KUKA KRL program: MyProgram_225().src

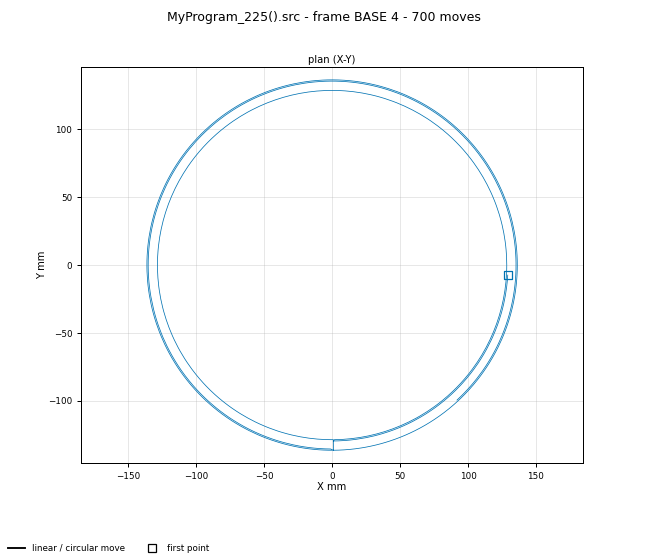
[picture p0: tool path of MyProgram_225().src in frame BASE 4, 700 of 700 moves have a stored position in this frame; points joined in program order, loops and branches not executed]
&ACCESS RVP
&REL 1
&PARAM TEMPLATE = C:\KRC\Roboter\Template\vorgabe
&PARAM EDITMASK = *
DEF MyProgram_225()
; ---- Setting reference (Base) ----
$BASE = BASE_DATA[4]

; --------------------------
; ---- Setting tool (TCP) ----
$TOOL = TOOL_DATA[3]
; --------------------------

$VEL.CP = VEL_APROX_PRINT
Startdeposition()
$VEL.CP = VEL_PRINT
LIN {X 129.2474,Y -7.3831,Z 155,A -4.9657,B 16.1496,C -0.2216,E1 16.3104,E2 814.1101} C_DIS
LIN {X 128.9531,Y -11.421,Z 155,A -6.9054,B 16.1497,C -0.211,E1 16.3099,E2 816.0693} C_DIS
LIN {X 128.4281,Y -16.2953,Z 155,A -8.4504,B 16.1495,C -0.2265,E1 16.3095,E2 817.5445} C_DIS
LIN {X 127.4709,Y -22.5885,Z 155,A -10.9683,B 16.1495,C -0.2286,E1 16.3084,E2 820.031} C_DIS
LIN {X 127.0051,Y -25.0853,Z 155,A -12.6562,B 16.1498,C -0.2051,E1 16.3075,E2 821.7867} C_DIS
LIN {X 126.3261,Y -28.3023,Z 155,A -13.8755,B 16.1498,C -0.2091,E1 16.3067,E2 822.9803} C_DIS
LIN {X 125.3243,Y -32.4531,Z 155,A -15.5909,B 16.1498,C -0.2097,E1 16.3056,E2 824.678} C_DIS
LIN {X 124.4903,Y -35.5191,Z 155,A -17.2829,B 16.1499,C -0.1954,E1 16.3043,E2 826.4054} C_DIS
LIN {X 122.9714,Y -40.4627,Z 155,A -19.3134,B 16.1499,C -0.1978,E1 16.3026,E2 828.4087} C_DIS
LIN {X 121.7271,Y -44.0625,Z 155,A -21.5995,B 16.1502,C -0.1717,E1 16.3004,E2 830.7672} C_DIS
LIN {X 119.9725,Y -48.6377,Z 155,A -23.157,B 16.15,C -0.187,E1 16.2988,E2 832.2564} C_DIS
LIN {X 118.5111,Y -52.1027,Z 155,A -24.7542,B 16.15,C -0.1846,E1 16.2971,E2 833.8481} C_DIS
LIN {X 117.1159,Y -55.1662,Z 155,A -26.2187,B 16.15,C -0.1813,E1 16.2954,E2 835.3116} C_DIS
LIN {X 114.7718,Y -59.8872,Z 155,A -28.3572,B 16.15,C -0.1817,E1 16.2927,E2 837.4305} C_DIS
LIN {X 113.6651,Y -61.9653,Z 155,A -29.6574,B 16.1502,C -0.1696,E1 16.2909,E2 838.7625} C_DIS
LIN {X 111.4503,Y -65.8666,Z 155,A -31.6784,B 16.1502,C -0.163,E1 16.2881,E2 840.7904} C_DIS
LIN {X 109.1625,Y -69.5921,Z 155,A -33.4546,B 16.1502,C -0.1634,E1 16.2855,E2 842.5506} C_DIS
LIN {X 107.339,Y -72.3729,Z 155,A -35.0483,B 16.1503,C -0.1553,E1 16.283,E2 844.1606} C_DIS
LIN {X 104.186,Y -76.8426,Z 155,A -37.4354,B 16.1503,C -0.1503,E1 16.2791,E2 846.547} C_DIS
LIN {X 101.853,Y -79.9088,Z 155,A -39.1319,B 16.1504,C -0.1463,E1 16.2762,E2 848.2447} C_DIS
LIN {X 99.343,Y -83.0089,Z 155,A -40.9388,B 16.1504,C -0.1406,E1 16.273,E2 850.0588} C_DIS
LIN {X 96.0502,Y -86.7978,Z 155,A -42.9236,B 16.1504,C -0.1435,E1 16.2694,E2 852.0187} C_DIS
LIN {X 93.7861,Y -89.2396,Z 155,A -44.5289,B 16.1505,C -0.1355,E1 16.2663,E2 853.6413} C_DIS
LIN {X 90.8438,Y -92.233,Z 155,A -46.4781,B 16.1505,C -0.1281,E1 16.2624,E2 855.6036} C_DIS
LIN {X 87.5864,Y -95.3314,Z 155,A -48.1246,B 16.1505,C -0.1357,E1 16.2591,E2 857.2121} C_DIS
LIN {X 85.2485,Y -97.4277,Z 155,A -49.6523,B 16.1505,C -0.1279,E1 16.2559,E2 858.7578} C_DIS
LIN {X 82.2321,Y -99.9874,Z 155,A -51.4278,B 16.1505,C -0.1234,E1 16.2521,E2 860.5383} C_DIS
LIN {X 78.358,Y -103.0515,Z 155,A -53.5577,B 16.1506,C -0.121,E1 16.2474,E2 862.6642} C_DIS
LIN {X 75.3005,Y -105.3056,Z 155,A -55.2753,B 16.1506,C -0.1165,E1 16.2435,E2 864.388} C_DIS
LIN {X 71.8133,Y -107.714,Z 155,A -57.181,B 16.1506,C -0.112,E1 16.2391,E2 866.2994} C_DIS
LIN {X 68.6345,Y -109.7672,Z 155,A -58.8635,B 16.1507,C -0.1088,E1 16.2351,E2 867.9846} C_DIS
LIN {X 64.898,Y -112.0165,Z 155,A -60.7724,B 16.1507,C -0.1063,E1 16.2305,E2 869.8931} C_DIS
LIN {X 59.3003,Y -115.0774,Z 155,A -63.965,B 16.1508,C -0.0893,E1 16.2226,E2 873.1319} C_DIS
LIN {X 55.719,Y -116.8518,Z 155,A -65.2781,B 16.1508,C -0.1022,E1 16.2194,E2 874.3933} C_DIS
LIN {X 52.249,Y -118.4459,Z 155,A -67.4256,B 16.1508,C -0.0844,E1 16.2138,E2 876.596} C_DIS
LIN {X 48.4916,Y -120.0314,Z 155,A -68.8253,B 16.1508,C -0.0957,E1 16.2103,E2 877.9501} C_DIS
LIN {X 45.0598,Y -121.3619,Z 155,A -70.3403,B 16.1508,C -0.0975,E1 16.2063,E2 879.4531} C_DIS
LIN {X 41.6197,Y -122.5861,Z 155,A -72.6412,B 16.1508,C -0.0727,E1 16.2001,E2 881.8356} C_DIS
LIN {X 36.809,Y -124.114,Z 155,A -74.0346,B 16.1508,C -0.0985,E1 16.1966,E2 883.1326} C_DIS
LIN {X 33.8596,Y -124.9512,Z 155,A -75.564,B 16.1508,C -0.0914,E1 16.1924,E2 884.6834} C_DIS
LIN {X 30.5927,Y -125.7901,Z 155,A -77.8519,B 16.1509,C -0.0637,E1 16.186,E2 887.0651} C_DIS
LIN {X 24.8487,Y -127.0506,Z 155,A -79.6789,B 16.1509,C -0.0873,E1 16.1812,E2 888.8038} C_DIS
LIN {X 17.4336,Y -128.279,Z 155,A -82.8576,B 16.1509,C -0.0901,E1 16.1725,E2 891.9675} C_DIS
LIN {X 13.1784,Y -128.786,Z 155,A -84.9822,B 16.1509,C -0.0816,E1 16.1665,E2 894.12} C_DIS
LIN {X 9.2675,Y -129.1248,Z 155,A -86.6956,B 16.1509,C -0.0817,E1 16.1617,E2 895.8316} C_DIS
LIN {X 4.804,Y -129.3679,Z 155,A -88.6412,B 16.1509,C -0.0822,E1 16.1563,E2 897.7745} C_DIS
LIN {X 0.918,Y -129.4524,Z 155,A -89.6672,B 16.1507,C -0.1046,E1 16.1537,E2 898.7195} C_DIS
Enddeposition()
LIN {X 0.918,Y -129.4524,Z 155,A -89.6672,B 16.1507,C -0.1046,E1 16.1537,E2 898.7195} C_DIS
Startdeposition()
$VEL.CP = VEL_PRINT
LIN {X 1.6778,Y -128.5115,Z 155,A -89.2328,B 16.1506,C -0.1179,E1 16.1549,E2 898.2373} C_DIS
LIN {X 4.7325,Y -128.4347,Z 155,A -87.9227,B 16.1506,C -0.1166,E1 16.1586,E2 896.9326} C_DIS
LIN {X 7.9871,Y -128.2732,Z 155,A -86.5233,B 16.1506,C -0.1153,E1 16.1625,E2 895.5387} C_DIS
LIN {X 11.132,Y -128.0389,Z 155,A -85.1192,B 16.1506,C -0.1158,E1 16.1664,E2 894.134} C_DIS
LIN {X 14.3466,Y -127.7196,Z 155,A -83.6808,B 16.1506,C -0.1165,E1 16.1704,E2 892.6949} C_DIS
LIN {X 17.4169,Y -127.3379,Z 155,A -82.2994,B 16.1506,C -0.1173,E1 16.1742,E2 891.3124} C_DIS
LIN {X 20.4129,Y -126.8922,Z 155,A -80.9516,B 16.1506,C -0.118,E1 16.1779,E2 889.964} C_DIS
LIN {X 23.6323,Y -126.331,Z 155,A -79.5141,B 16.1506,C -0.1184,E1 16.1819,E2 888.5277} C_DIS
LIN {X 26.7059,Y -125.7168,Z 155,A -78.0866,B 16.1506,C -0.1205,E1 16.1858,E2 887.0956} C_DIS
LIN {X 30.0992,Y -124.947,Z 155,A -76.4897,B 16.1506,C -0.1234,E1 16.1902,E2 885.4921} C_DIS
LIN {X 32.8535,Y -124.2515,Z 155,A -75.2461,B 16.1506,C -0.1238,E1 16.1935,E2 884.2502} C_DIS
LIN {X 35.7824,Y -123.4401,Z 155,A -73.9279,B 16.1506,C -0.1238,E1 16.197,E2 882.9352} C_DIS
LIN {X 38.7952,Y -122.5265,Z 155,A -72.5303,B 16.1506,C -0.1252,E1 16.2008,E2 881.537} C_DIS
LIN {X 42.2001,Y -121.3954,Z 155,A -71.0011,B 16.1506,C -0.1246,E1 16.2048,E2 880.0147} C_DIS
LIN {X 44.8787,Y -120.431,Z 155,A -69.6719,B 16.1505,C -0.1282,E1 16.2083,E2 878.6774} C_DIS
LIN {X 47.8161,Y -119.2953,Z 155,A -68.2677,B 16.1505,C -0.13,E1 16.212,E2 877.2717} C_DIS
LIN {X 50.745,Y -118.0792,Z 155,A -66.9012,B 16.1505,C -0.1302,E1 16.2155,E2 875.9094} C_DIS
LIN {X 53.6147,Y -116.8044,Z 155,A -65.477,B 16.1505,C -0.133,E1 16.2191,E2 874.481} C_DIS
LIN {X 56.4616,Y -115.4553,Z 155,A -64.0855,B 16.1505,C -0.1346,E1 16.2226,E2 873.0897} C_DIS
LIN {X 59.1544,Y -114.1002,Z 155,A -62.7618,B 16.1505,C -0.136,E1 16.2259,E2 871.767} C_DIS
LIN {X 61.9121,Y -112.6286,Z 155,A -61.238,B 16.1504,C -0.1427,E1 16.2297,E2 870.2265} C_DIS
LIN {X 64.7163,Y -111.041,Z 155,A -59.8975,B 16.1504,C -0.1417,E1 16.2329,E2 868.8957} C_DIS
LIN {X 67.5215,Y -109.3579,Z 155,A -58.4653,B 16.1504,C -0.1433,E1 16.2363,E2 867.4651} C_DIS
LIN {X 70.18,Y -107.6707,Z 155,A -57.0713,B 16.1504,C -0.1455,E1 16.2396,E2 866.0706} C_DIS
LIN {X 72.7088,Y -105.9792,Z 155,A -55.7279,B 16.1504,C -0.1476,E1 16.2427,E2 864.7272} C_DIS
LIN {X 75.3703,Y -104.1032,Z 155,A -54.2861,B 16.1504,C -0.15,E1 16.2459,E2 863.2849} C_DIS
LIN {X 78.4386,Y -101.812,Z 155,A -52.4335,B 16.1502,C -0.1584,E1 16.2501,E2 861.4131} C_DIS
LIN {X 81.5351,Y -99.3492,Z 155,A -50.6751,B 16.1502,C -0.1618,E1 16.2539,E2 859.6532} C_DIS
LIN {X 85.1286,Y -96.2875,Z 155,A -48.5905,B 16.1502,C -0.1656,E1 16.2583,E2 857.5684} C_DIS
LIN {X 88.6071,Y -93.0967,Z 155,A -46.5125,B 16.1502,C -0.1692,E1 16.2626,E2 855.4909} C_DIS
LIN {X 91.4722,Y -90.2838,Z 155,A -44.7234,B 16.1501,C -0.1733,E1 16.2661,E2 853.6997} C_DIS
LIN {X 94.6884,Y -86.9039,Z 155,A -42.6573,B 16.1501,C -0.1776,E1 16.27,E2 851.6326} C_DIS
LIN {X 97.8259,Y -83.3563,Z 155,A -40.5635,B 16.15,C -0.1821,E1 16.2739,E2 849.5381} C_DIS
LIN {X 100.8306,Y -79.6963,Z 155,A -38.4709,B 16.15,C -0.1866,E1 16.2775,E2 847.445} C_DIS
LIN {X 103.2224,Y -76.5725,Z 155,A -36.8644,B 16.15,C -0.1858,E1 16.2802,E2 845.8536} C_DIS
LIN {X 105.4013,Y -73.5443,Z 155,A -35.3387,B 16.15,C -0.1853,E1 16.2827,E2 844.3419} C_DIS
LIN {X 106.8625,Y -71.4043,Z 155,A -34.0899,B 16.1499,C -0.1916,E1 16.2846,E2 843.0805} C_DIS
LIN {X 108.5817,Y -68.7621,Z 155,A -32.6993,B 16.1499,C -0.1948,E1 16.2867,E2 841.6896} C_DIS
LIN {X 110.2875,Y -65.9916,Z 155,A -31.1326,B 16.1498,C -0.2028,E1 16.289,E2 840.1073} C_DIS
LIN {X 111.8819,Y -63.2511,Z 155,A -29.8604,B 16.1498,C -0.2016,E1 16.2908,E2 838.8498} C_DIS
LIN {X 113.3987,Y -60.4901,Z 155,A -28.4494,B 16.1498,C -0.2057,E1 16.2926,E2 837.4361} C_DIS
LIN {X 114.8075,Y -57.769,Z 155,A -27.1034,B 16.1497,C -0.2088,E1 16.2943,E2 836.0906} C_DIS
LIN {X 116.1854,Y -54.9443,Z 155,A -25.6971,B 16.1497,C -0.2129,E1 16.296,E2 834.6817} C_DIS
LIN {X 117.4948,Y -52.0848,Z 155,A -24.329,B 16.1496,C -0.2157,E1 16.2976,E2 833.3156} C_DIS
LIN {X 118.734,Y -49.194,Z 155,A -22.9407,B 16.1496,C -0.2192,E1 16.2991,E2 831.927} C_DIS
LIN {X 119.9017,Y -46.2748,Z 155,A -21.5531,B 16.1495,C -0.2228,E1 16.3005,E2 830.5392} C_DIS
LIN {X 121.0454,Y -43.1959,Z 155,A -20.102,B 16.1495,C -0.2266,E1 16.3019,E2 829.0876} C_DIS
LIN {X 122.0688,Y -40.2129,Z 155,A -18.7106,B 16.1494,C -0.2302,E1 16.3031,E2 827.696} C_DIS
LIN {X 123.0231,Y -37.1916,Z 155,A -17.3224,B 16.1494,C -0.2335,E1 16.3043,E2 826.3087} C_DIS
LIN {X 123.8678,Y -34.2723,Z 155,A -15.9674,B 16.1493,C -0.2375,E1 16.3053,E2 824.9518} C_DIS
LIN {X 124.6966,Y -31.1243,Z 155,A -14.5432,B 16.1493,C -0.2409,E1 16.3063,E2 823.5288} C_DIS
LIN {X 125.398,Y -28.1654,Z 155,A -13.1855,B 16.1492,C -0.245,E1 16.3072,E2 822.169} C_DIS
LIN {X 126.0535,Y -25.0714,Z 155,A -11.7956,B 16.1492,C -0.2485,E1 16.3079,E2 820.7795} C_DIS
LIN {X 126.6293,Y -21.9819,Z 155,A -10.4121,B 16.1491,C -0.2521,E1 16.3086,E2 819.3962} C_DIS
LIN {X 127.1333,Y -18.8507,Z 155,A -8.9602,B 16.149,C -0.2578,E1 16.3092,E2 817.9379} C_DIS
LIN {X 127.5546,Y -15.7436,Z 155,A -7.5816,B 16.149,C -0.2613,E1 16.3097,E2 816.5597} C_DIS
LIN {X 127.9003,Y -12.6262,Z 155,A -6.2052,B 16.1489,C -0.2648,E1 16.3101,E2 815.184} C_DIS
LIN {X 128.1695,Y -9.507,Z 155,A -4.852,B 16.1489,C -0.2676,E1 16.3104,E2 813.8339} C_DIS
LIN {X 128.3721,Y -6.2015,Z 155,A -3.3818,B 16.1488,C -0.2718,E1 16.3107,E2 812.3625} C_DIS
LIN {X 128.4838,Y -3.1456,Z 155,A -2.0505,B 16.1488,C -0.2748,E1 16.3107,E2 811.0332} C_DIS
LIN {X 128.5245,Y 0.0068,Z 155,A -0.4873,B 16.1486,C -0.2847,E1 16.3107,E2 809.4497} C_DIS
LIN {X 128.4806,Y 3.2619,Z 155,A 0.7946,B 16.1486,C -0.2831,E1 16.3107,E2 808.1858} C_DIS
LIN {X 128.3589,Y 6.4648,Z 155,A 2.2721,B 16.1485,C -0.2892,E1 16.3105,E2 806.7007} C_DIS
LIN {X 128.0428,Y 11.0858,Z 155,A 4.2244,B 16.1485,C -0.2914,E1 16.3101,E2 804.7591} C_DIS
LIN {X 127.7458,Y 14.1038,Z 155,A 5.7395,B 16.1483,C -0.3013,E1 16.3097,E2 803.2231} C_DIS
LIN {X 127.3364,Y 17.4282,Z 155,A 7.0732,B 16.1483,C -0.3001,E1 16.3092,E2 801.9065} C_DIS
LIN {X 126.8629,Y 20.5886,Z 155,A 8.5421,B 16.1482,C -0.3059,E1 16.3085,E2 800.4307} C_DIS
LIN {X 126.3334,Y 23.6197,Z 155,A 9.8059,B 16.1482,C -0.3062,E1 16.3079,E2 799.1778} C_DIS
LIN {X 125.7187,Y 26.6971,Z 155,A 11.225,B 16.1481,C -0.311,E1 16.3071,E2 797.7547} C_DIS
LIN {X 125.0528,Y 29.6603,Z 155,A 12.6772,B 16.1479,C -0.3185,E1 16.3062,E2 796.2895} C_DIS
LIN {X 124.0111,Y 33.7549,Z 155,A 14.5681,B 16.1479,C -0.3242,E1 16.3048,E2 794.3957} C_DIS
LIN {X 122.9892,Y 37.3025,Z 155,A 16.0644,B 16.1479,C -0.3237,E1 16.3037,E2 792.915} C_DIS
LIN {X 122.0342,Y 40.3168,Z 155,A 17.4933,B 16.1477,C -0.3284,E1 16.3024,E2 791.4823} C_DIS
LIN {X 120.9718,Y 43.3998,Z 155,A 18.8986,B 16.1477,C -0.3308,E1 16.3011,E2 790.0811} C_DIS
LIN {X 119.8705,Y 46.3552,Z 155,A 20.2903,B 16.1477,C -0.3342,E1 16.2997,E2 788.6896} C_DIS
LIN {X 118.397,Y 50.001,Z 155,A 22.1728,B 16.1474,C -0.3436,E1 16.2977,E2 786.7902} C_DIS
LIN {X 116.81,Y 53.6026,Z 155,A 23.7609,B 16.1474,C -0.3425,E1 16.2959,E2 785.2198} C_DIS
LIN {X 115.4748,Y 56.4221,Z 155,A 25.2247,B 16.1474,C -0.3488,E1 16.2941,E2 783.7462} C_DIS
LIN {X 114.0834,Y 59.1864,Z 155,A 26.4948,B 16.1474,C -0.3486,E1 16.2925,E2 782.4876} C_DIS
LIN {X 112.594,Y 61.9747,Z 155,A 27.9079,B 16.1473,C -0.3525,E1 16.2906,E2 781.0728} C_DIS
LIN {X 111.041,Y 64.7163,Z 155,A 29.3254,B 16.1472,C -0.3565,E1 16.2887,E2 779.6526} C_DIS
LIN {X 109.0767,Y 67.9739,Z 155,A 30.8966,B 16.1472,C -0.3565,E1 16.2864,E2 778.0945} C_DIS
LIN {X 107.6796,Y 70.1663,Z 155,A 32.139,B 16.147,C -0.3623,E1 16.2845,E2 776.8415} C_DIS
LIN {X 106.0025,Y 72.6749,Z 155,A 33.4662,B 16.147,C -0.3649,E1 16.2824,E2 775.5152} C_DIS
LIN {X 104.1598,Y 75.2922,Z 155,A 35.0142,B 16.1468,C -0.3726,E1 16.2799,E2 773.9521} C_DIS
LIN {X 101.8049,Y 78.4478,Z 155,A 36.7885,B 16.1468,C -0.3773,E1 16.2769,E2 772.1743} C_DIS
LIN {X 99.345,Y 81.5402,Z 155,A 38.5399,B 16.1466,C -0.381,E1 16.2738,E2 770.4229} C_DIS
LIN {X 96.7667,Y 84.5835,Z 155,A 40.291,B 16.1466,C -0.384,E1 16.2706,E2 768.6738} C_DIS
LIN {X 94.1318,Y 87.5065,Z 155,A 42.0259,B 16.1465,C -0.3872,E1 16.2673,E2 766.94} C_DIS
LIN {X 90.9193,Y 90.8404,Z 155,A 43.9575,B 16.1465,C -0.3869,E1 16.2636,E2 765.0225} C_DIS
LIN {X 88.0408,Y 93.6324,Z 155,A 45.8629,B 16.1463,C -0.3946,E1 16.2597,E2 763.1025} C_DIS
LIN {X 85.1331,Y 96.2835,Z 155,A 47.6115,B 16.1463,C -0.3978,E1 16.2561,E2 761.3538} C_DIS
LIN {X 81.5387,Y 99.3462,Z 155,A 49.7011,B 16.1461,C -0.4012,E1 16.2516,E2 759.265} C_DIS
LIN {X 77.8639,Y 102.2519,Z 155,A 51.7741,B 16.1461,C -0.4043,E1 16.247,E2 757.193} C_DIS
LIN {X 75.2011,Y 104.2259,Z 155,A 53.1006,B 16.1461,C -0.4017,E1 16.2441,E2 755.8833} C_DIS
LIN {X 72.7118,Y 105.9772,Z 155,A 54.4455,B 16.1461,C -0.4036,E1 16.241,E2 754.5394} C_DIS
LIN {X 70.092,Y 107.7279,Z 155,A 55.8445,B 16.1461,C -0.4056,E1 16.2377,E2 753.1406} C_DIS
LIN {X 67.1684,Y 109.5745,Z 155,A 57.3256,B 16.1461,C -0.4059,E1 16.2342,E2 751.666} C_DIS
LIN {X 64.6725,Y 111.0664,Z 155,A 58.6546,B 16.146,C -0.4089,E1 16.231,E2 750.3329} C_DIS
LIN {X 61.9909,Y 112.585,Z 155,A 60.0556,B 16.1459,C -0.4117,E1 16.2276,E2 748.9285} C_DIS
LIN {X 59.1897,Y 114.0817,Z 155,A 61.4531,B 16.1459,C -0.4129,E1 16.2241,E2 747.5329} C_DIS
LIN {X 56.3717,Y 115.4997,Z 155,A 62.8516,B 16.1459,C -0.4144,E1 16.2206,E2 746.1351} C_DIS
LIN {X 53.4283,Y 116.8906,Z 155,A 64.4625,B 16.1456,C -0.4215,E1 16.2165,E2 744.5056} C_DIS
LIN {X 50.3552,Y 118.2477,Z 155,A 65.7823,B 16.1457,C -0.4172,E1 16.2132,E2 743.2063} C_DIS
LIN {X 47.7503,Y 119.3218,Z 155,A 67.0354,B 16.1457,C -0.4184,E1 16.2099,E2 741.9534} C_DIS
LIN {X 44.849,Y 120.4422,Z 155,A 68.4256,B 16.1457,C -0.4199,E1 16.2063,E2 740.5628} C_DIS
LIN {X 41.711,Y 121.565,Z 155,A 69.9001,B 16.1457,C -0.4208,E1 16.2024,E2 739.0897} C_DIS
LIN {X 38.7098,Y 122.5538,Z 155,A 71.3037,B 16.1457,C -0.4218,E1 16.1987,E2 737.6867} C_DIS
LIN {X 35.5655,Y 123.5035,Z 155,A 72.7486,B 16.1457,C -0.4223,E1 16.1948,E2 736.2442} C_DIS
LIN {X 32.2348,Y 124.4148,Z 155,A 74.4562,B 16.1455,C -0.4289,E1 16.1902,E2 734.5175} C_DIS
LIN {X 28.1665,Y 125.3977,Z 155,A 76.1659,B 16.1455,C -0.4249,E1 16.1856,E2 732.826} C_DIS
LIN {X 25.0874,Y 126.0502,Z 155,A 77.5622,B 16.1455,C -0.4253,E1 16.1818,E2 731.4308} C_DIS
LIN {X 21.9616,Y 126.633,Z 155,A 78.9684,B 16.1455,C -0.4256,E1 16.1779,E2 730.0263} C_DIS
LIN {X 18.8606,Y 127.1318,Z 155,A 80.4238,B 16.1455,C -0.4279,E1 16.1739,E2 728.5649} C_DIS
LIN {X 15.7531,Y 127.5535,Z 155,A 81.8154,B 16.1455,C -0.4281,E1 16.17,E2 727.1745} C_DIS
LIN {X 12.6343,Y 127.8995,Z 155,A 83.2064,B 16.1455,C -0.4281,E1 16.1662,E2 725.7848} C_DIS
LIN {X 9.5076,Y 128.1695,Z 155,A 84.6793,B 16.1455,C -0.4307,E1 16.162,E2 724.304} C_DIS
LIN {X 4.7612,Y 128.4336,Z 155,A 86.6769,B 16.1455,C -0.4268,E1 16.1565,E2 722.3212} C_DIS
LIN {X 1.5922,Y 128.5129,Z 155,A 88.0233,B 16.1455,C -0.4246,E1 16.1528,E2 720.9832} C_DIS
LIN {X -1.6807,Y 128.5115,Z 155,A 89.5801,B 16.1455,C -0.4276,E1 16.1484,E2 719.4159} C_DIS
LIN {X -4.7248,Y 128.435,Z 155,A 91.0568,B 16.1454,C -0.4311,E1 16.1442,E2 717.9262} C_DIS
LIN {X -8.3936,Y 128.2481,Z 155,A 92.51,B 16.1456,C -0.4248,E1 16.1402,E2 716.495} C_DIS
LIN {X -11.1743,Y 128.0353,Z 155,A 93.7856,B 16.1456,C -0.4254,E1 16.1367,E2 715.2165} C_DIS
LIN {X -14.2979,Y 127.7249,Z 155,A 95.1896,B 16.1456,C -0.4249,E1 16.1328,E2 713.8128} C_DIS
LIN {X -17.4144,Y 127.3382,Z 155,A 96.7612,B 16.1454,C -0.4296,E1 16.1284,E2 712.2225} C_DIS
LIN {X -20.5195,Y 126.8744,Z 155,A 98.0601,B 16.1455,C -0.4256,E1 16.1248,E2 710.9361} C_DIS
LIN {X -23.6138,Y 126.3345,Z 155,A 99.3856,B 16.1456,C -0.4224,E1 16.1212,E2 709.62} C_DIS
LIN {X -26.7229,Y 125.7131,Z 155,A 100.8372,B 16.1456,C -0.4226,E1 16.1172,E2 708.1651} C_DIS
LIN {X -29.6889,Y 125.0459,Z 155,A 102.2295,B 16.1456,C -0.4226,E1 16.1134,E2 706.7697} C_DIS
LIN {X -32.86,Y 124.2498,Z 155,A 103.6553,B 16.1456,C -0.4204,E1 16.1096,E2 705.3486} C_DIS
LIN {X -35.7921,Y 123.4372,Z 155,A 105.0154,B 16.1456,C -0.4192,E1 16.1059,E2 703.9891} C_DIS
LIN {X -38.806,Y 122.523,Z 155,A 106.4232,B 16.1457,C -0.418,E1 16.1022,E2 702.5821} C_DIS
LIN {X -41.7983,Y 121.5348,Z 155,A 107.8642,B 16.1457,C -0.4176,E1 16.0984,E2 701.1382} C_DIS
LIN {X -44.8793,Y 120.4308,Z 155,A 109.2974,B 16.1458,C -0.4151,E1 16.0946,E2 699.7092} C_DIS
LIN {X -47.8351,Y 119.2876,Z 155,A 110.714,B 16.1458,C -0.4135,E1 16.0909,E2 698.2935} C_DIS
LIN {X -50.7426,Y 118.0802,Z 155,A 112.09,B 16.1459,C -0.4109,E1 16.0874,E2 696.922} C_DIS
LIN {X -53.6201,Y 116.8019,Z 155,A 113.6569,B 16.1459,C -0.4139,E1 16.0834,E2 695.3378} C_DIS
LIN {X -56.4654,Y 115.4535,Z 155,A 114.9395,B 16.1459,C -0.4083,E1 16.0802,E2 694.0705} C_DIS
LIN {X -59.1815,Y 114.086,Z 155,A 116.283,B 16.146,C -0.4059,E1 16.0769,E2 692.7297} C_DIS
LIN {X -61.9561,Y 112.6043,Z 155,A 117.7111,B 16.146,C -0.4045,E1 16.0734,E2 691.3001} C_DIS
LIN {X -65.2941,Y 110.7019,Z 155,A 119.334,B 16.1462,C -0.399,E1 16.0695,E2 689.6892} C_DIS
LIN {X -67.5233,Y 109.3567,Z 155,A 120.6102,B 16.1462,C -0.4005,E1 16.0664,E2 688.4012} C_DIS
LIN {X -70.1807,Y 107.6703,Z 155,A 122.0204,B 16.1462,C -0.3983,E1 16.0631,E2 686.9917} C_DIS
LIN {X -72.7105,Y 105.9781,Z 155,A 123.3807,B 16.1462,C -0.396,E1 16.0599,E2 685.6326} C_DIS
LIN {X -75.3746,Y 104.1001,Z 155,A 124.8414,B 16.1463,C -0.3935,E1 16.0566,E2 684.1726} C_DIS
LIN {X -78.4549,Y 101.7994,Z 155,A 126.7263,B 16.1463,C -0.3953,E1 16.0524,E2 682.2702} C_DIS
LIN {X -82.1023,Y 98.8807,Z 155,A 128.6844,B 16.1465,C -0.3874,E1 16.0482,E2 680.3288} C_DIS
LIN {X -85.1338,Y 96.2829,Z 155,A 130.6129,B 16.1465,C -0.3882,E1 16.0441,E2 678.3855} C_DIS
LIN {X -88.616,Y 93.0883,Z 155,A 132.7189,B 16.1465,C -0.3836,E1 16.0398,E2 676.2821} C_DIS
LIN {X -91.4742,Y 90.2818,Z 155,A 134.533,B 16.1466,C -0.3804,E1 16.0362,E2 674.4671} C_DIS
LIN {X -94.6944,Y 86.8973,Z 155,A 136.6338,B 16.1467,C -0.3762,E1 16.0322,E2 672.3668} C_DIS
LIN {X -97.8335,Y 83.3474,Z 155,A 138.7579,B 16.1468,C -0.3715,E1 16.0283,E2 670.2442} C_DIS
LIN {X -100.8339,Y 79.6922,Z 155,A 140.8828,B 16.1469,C -0.3669,E1 16.0246,E2 668.1201} C_DIS
LIN {X -103.6736,Y 75.9603,Z 155,A 142.9652,B 16.1471,C -0.3614,E1 16.0211,E2 666.0414} C_DIS
LIN {X -105.981,Y 72.7062,Z 155,A 144.6287,B 16.1472,C -0.3535,E1 16.0185,E2 664.3933} C_DIS
LIN {X -107.7317,Y 70.0861,Z 155,A 146.0428,B 16.1472,C -0.3501,E1 16.0163,E2 662.98} C_DIS
LIN {X -109.4371,Y 67.3924,Z 155,A 147.5003,B 16.1474,C -0.3474,E1 16.0142,E2 661.5204} C_DIS
LIN {X -111.0995,Y 64.6152,Z 155,A 148.9274,B 16.1474,C -0.3431,E1 16.0122,E2 660.097} C_DIS
LIN {X -112.6399,Y 61.8916,Z 155,A 150.3436,B 16.1475,C -0.3399,E1 16.0102,E2 658.6802} C_DIS
LIN {X -114.0659,Y 59.2198,Z 155,A 151.7105,B 16.1475,C -0.3367,E1 16.0085,E2 657.3133} C_DIS
LIN {X -115.472,Y 56.4279,Z 155,A 153.1143,B 16.1476,C -0.3332,E1 16.0067,E2 655.9101} C_DIS
LIN {X -116.9071,Y 53.3926,Z 155,A 154.6176,B 16.1477,C -0.3292,E1 16.005,E2 654.4082} C_DIS
LIN {X -118.1251,Y 50.6389,Z 155,A 155.978,B 16.1477,C -0.3259,E1 16.0034,E2 653.0476} C_DIS
LIN {X -119.3315,Y 47.7262,Z 155,A 157.3951,B 16.1479,C -0.3222,E1 16.002,E2 651.631} C_DIS
LIN {X -120.4648,Y 44.7886,Z 155,A 158.9725,B 16.1479,C -0.3232,E1 16.0004,E2 650.0357} C_DIS
LIN {X -121.571,Y 41.6936,Z 155,A 160.2898,B 16.148,C -0.3146,E1 15.9992,E2 648.7374} C_DIS
LIN {X -122.5556,Y 38.7039,Z 155,A 161.7056,B 16.148,C -0.3109,E1 15.998,E2 647.322} C_DIS
LIN {X -123.4378,Y 35.7902,Z 155,A 163.0752,B 16.1481,C -0.3072,E1 15.9969,E2 645.9529} C_DIS
LIN {X -124.2779,Y 32.7544,Z 155,A 164.5019,B 16.1482,C -0.3037,E1 15.9959,E2 644.5255} C_DIS
LIN {X -125.0663,Y 29.6042,Z 155,A 165.9454,B 16.1482,C -0.2993,E1 15.9949,E2 643.0846} C_DIS
LIN {X -125.7594,Y 26.5087,Z 155,A 167.3726,B 16.1484,C -0.2954,E1 15.9941,E2 641.6577} C_DIS
LIN {X -126.3736,Y 23.4092,Z 155,A 168.7947,B 16.1484,C -0.2916,E1 15.9933,E2 640.2361} C_DIS
LIN {X -126.8922,Y 20.413,Z 155,A 170.187,B 16.1484,C -0.2885,E1 15.9927,E2 638.8414} C_DIS
LIN {X -127.3673,Y 17.1922,Z 155,A 171.6167,B 16.1486,C -0.2835,E1 15.9921,E2 637.416} C_DIS
LIN {X -127.7498,Y 14.0661,Z 155,A 173.0367,B 16.1486,C -0.2797,E1 15.9917,E2 635.9961} C_DIS
LIN {X -128.0558,Y 10.9315,Z 155,A 174.5773,B 16.1486,C -0.2794,E1 15.9913,E2 634.4417} C_DIS
LIN {X -128.3723,Y 6.1984,Z 155,A 176.6048,B 16.1488,C -0.2705,E1 15.9909,E2 632.427} C_DIS
LIN {X -128.4839,Y 3.1442,Z 155,A 177.9794,B 16.1488,C -0.2667,E1 15.9909,E2 631.0528} C_DIS
LIN {X -128.5227,Y -0.3076,Z 155,A 179.5287,B 16.1489,C -0.2623,E1 15.9908,E2 629.5043} C_DIS
LIN {X -128.4808,Y -3.2555,Z 155,A -179.1131,B 16.1489,C -0.2596,E1 15.9908,E2 628.1427} C_DIS
LIN {X -128.3613,Y -6.4158,Z 155,A -177.7056,B 16.149,C -0.2552,E1 15.991,E2 626.7373} C_DIS
LIN {X -128.1736,Y -9.4516,Z 155,A -176.3245,B 16.149,C -0.2519,E1 15.9913,E2 625.355} C_DIS
LIN {X -127.9039,Y -12.5881,Z 155,A -174.9169,B 16.1491,C -0.2478,E1 15.9917,E2 623.9487} C_DIS
LIN {X -127.5551,Y -15.7397,Z 155,A -173.4977,B 16.1492,C -0.2437,E1 15.9921,E2 622.5306} C_DIS
LIN {X -127.1162,Y -18.9666,Z 155,A -172.013,B 16.1492,C -0.2403,E1 15.9927,E2 621.0439} C_DIS
LIN {X -126.5619,Y -22.3588,Z 155,A -170.565,B 16.1494,C -0.2333,E1 15.9934,E2 619.6074} C_DIS
LIN {X -126.0547,Y -25.0654,Z 155,A -169.1982,B 16.1494,C -0.2337,E1 15.9941,E2 618.226} C_DIS
LIN {X -125.3178,Y -28.5165,Z 155,A -167.7516,B 16.1494,C -0.2254,E1 15.995,E2 616.7957} C_DIS
LIN {X -124.6437,Y -31.3329,Z 155,A -166.3438,B 16.1494,C -0.225,E1 15.9959,E2 615.376} C_DIS
LIN {X -123.8379,Y -34.3794,Z 155,A -164.956,B 16.1495,C -0.2205,E1 15.9969,E2 613.9918} C_DIS
LIN {X -122.8127,Y -37.8792,Z 155,A -163.3461,B 16.1495,C -0.2153,E1 15.9982,E2 612.3855} C_DIS
LIN {X -122.0281,Y -40.335,Z 155,A -162.1281,B 16.1496,C -0.2141,E1 15.9993,E2 611.1608} C_DIS
LIN {X -120.9675,Y -43.4119,Z 155,A -160.664,B 16.1496,C -0.2104,E1 16.0006,E2 609.6967} C_DIS
LIN {X -119.8681,Y -46.3612,Z 155,A -159.2486,B 16.1497,C -0.2068,E1 16.002,E2 608.2813} C_DIS
LIN {X -118.6967,Y -49.2832,Z 155,A -157.8335,B 16.1497,C -0.2033,E1 16.0035,E2 606.8663} C_DIS
LIN {X -117.4977,Y -52.0782,Z 155,A -156.4353,B 16.1497,C -0.2008,E1 16.0051,E2 605.4646} C_DIS
LIN {X -116.1416,Y -55.036,Z 155,A -154.8888,B 16.1497,C -0.1997,E1 16.0069,E2 603.9084} C_DIS
LIN {X -114.683,Y -58.0135,Z 155,A -153.6047,B 16.1499,C -0.1901,E1 16.0085,E2 602.6481} C_DIS
LIN {X -113.3465,Y -60.5873,Z 155,A -152.0805,B 16.1499,C -0.1935,E1 16.0105,E2 601.0984} C_DIS
LIN {X -111.8206,Y -63.3597,Z 155,A -150.7845,B 16.1499,C -0.1865,E1 16.0123,E2 599.817} C_DIS
LIN {X -109.9565,Y -66.5412,Z 155,A -149.236,B 16.15,C -0.1795,E1 16.0145,E2 598.2808} C_DIS
LIN {X -108.5292,Y -68.8451,Z 155,A -147.903,B 16.15,C -0.1802,E1 16.0165,E2 596.9345} C_DIS
LIN {X -106.8119,Y -71.4801,Z 155,A -146.5086,B 16.15,C -0.1765,E1 16.0186,E2 595.5421} C_DIS
LIN {X -104.7472,Y -74.4735,Z 155,A -144.9324,B 16.1501,C -0.1713,E1 16.0211,E2 593.9724} C_DIS
LIN {X -103.1677,Y -76.646,Z 155,A -143.5253,B 16.1501,C -0.1747,E1 16.0235,E2 592.5419} C_DIS
LIN {X -100.3591,Y -80.289,Z 155,A -141.428,B 16.1501,C -0.1714,E1 16.0271,E2 590.4406} C_DIS
LIN {X -97.7984,Y -83.3887,Z 155,A -139.6308,B 16.1501,C -0.1675,E1 16.0304,E2 588.6441} C_DIS
LIN {X -94.7032,Y -86.8877,Z 155,A -137.5307,B 16.1501,C -0.1636,E1 16.0343,E2 586.5433} C_DIS
LIN {X -92.5462,Y -89.1821,Z 155,A -136.1458,B 16.1502,C -0.1601,E1 16.037,E2 585.1615} C_DIS
LIN {X -89.7134,Y -92.0317,Z 155,A -134.311,B 16.1502,C -0.1577,E1 16.0406,E2 583.3226} C_DIS
LIN {X -86.3498,Y -95.1939,Z 155,A -132.3861,B 16.1503,C -0.1497,E1 16.0445,E2 581.4143} C_DIS
LIN {X -83.3528,Y -97.8289,Z 155,A -130.4506,B 16.1503,C -0.1511,E1 16.0486,E2 579.4614} C_DIS
LIN {X -79.6918,Y -100.8342,Z 155,A -128.3285,B 16.1503,C -0.1477,E1 16.0533,E2 577.339} C_DIS
LIN {X -76.5638,Y -103.2289,Z 155,A -126.6979,B 16.1503,C -0.1408,E1 16.0569,E2 575.7237} C_DIS
LIN {X -73.9209,Y -105.1375,Z 155,A -125.1567,B 16.1503,C -0.1412,E1 16.0604,E2 574.1728} C_DIS
LIN {X -70.4612,Y -107.487,Z 155,A -123.2631,B 16.1504,C -0.1392,E1 16.0648,E2 572.2764} C_DIS
LIN {X -67.4398,Y -109.408,Z 155,A -121.7569,B 16.1504,C -0.134,E1 16.0683,E2 570.7811} C_DIS
LIN {X -64.6643,Y -111.0711,Z 155,A -120.3202,B 16.1504,C -0.1318,E1 16.0718,E2 569.3454} C_DIS
LIN {X -61.8775,Y -112.6476,Z 155,A -118.8953,B 16.1504,C -0.1298,E1 16.0753,E2 567.9211} C_DIS
LIN {X -59.1892,Y -114.082,Z 155,A -117.5243,B 16.1504,C -0.1285,E1 16.0787,E2 566.5488} C_DIS
LIN {X -56.3757,Y -115.4977,Z 155,A -116.0511,B 16.1504,C -0.129,E1 16.0824,E2 565.0678} C_DIS
LIN {X -53.1312,Y -117.0267,Z 155,A -114.4209,B 16.1504,C -0.1281,E1 16.0865,E2 563.434} C_DIS
LIN {X -49.2123,Y -118.7263,Z 155,A -112.6061,B 16.1505,C -0.1233,E1 16.0911,E2 561.6297} C_DIS
LIN {X -46.3133,Y -119.8867,Z 155,A -111.2016,B 16.1505,C -0.1224,E1 16.0948,E2 560.2238} C_DIS
LIN {X -43.1996,Y -121.044,Z 155,A -109.7237,B 16.1505,C -0.121,E1 16.0987,E2 558.7462} C_DIS
LIN {X -40.2145,Y -122.0683,Z 155,A -108.2962,B 16.1505,C -0.1205,E1 16.1025,E2 557.3163} C_DIS
LIN {X -37.2017,Y -123.02,Z 155,A -106.8471,B 16.1505,C -0.1207,E1 16.1063,E2 555.8624} C_DIS
LIN {X -33.3267,Y -124.1253,Z 155,A -104.9818,B 16.1505,C -0.1217,E1 16.1114,E2 553.9887} C_DIS
LIN {X -29.7061,Y -125.0418,Z 155,A -103.4385,B 16.1505,C -0.1169,E1 16.1155,E2 552.4594} C_DIS
LIN {X -26.5311,Y -125.7545,Z 155,A -101.9934,B 16.1505,C -0.116,E1 16.1195,E2 551.0147} C_DIS
LIN {X -23.4153,Y -126.3725,Z 155,A -100.5753,B 16.1505,C -0.1155,E1 16.1234,E2 549.5961} C_DIS
LIN {X -20.4381,Y -126.888,Z 155,A -99.2173,B 16.1505,C -0.1154,E1 16.1271,E2 548.2364} C_DIS
LIN {X -17.2436,Y -127.3606,Z 155,A -97.6719,B 16.1505,C -0.1184,E1 16.1314,E2 546.6782} C_DIS
LIN {X -14.1435,Y -127.7415,Z 155,A -96.4122,B 16.1506,C -0.1139,E1 16.1349,E2 545.4336} C_DIS
LIN {X -10.9277,Y -128.0562,Z 155,A -94.9581,B 16.1506,C -0.1142,E1 16.1389,E2 543.9772} C_DIS
LIN {X -7.8771,Y -128.2799,Z 155,A -93.5617,B 16.1506,C -0.1152,E1 16.1428,E2 542.5765} C_DIS
LIN {X -4.7312,Y -128.4348,Z 155,A -92.1838,B 16.1506,C -0.1144,E1 16.1467,E2 541.2011} C_DIS
LIN {X -1.4707,Y -128.5149,Z 155,A -90.7474,B 16.1506,C -0.1139,E1 16.1507,E2 539.7661} C_DIS
LIN {X 0.9113,Y -128.517,Z 155,A -89.9648,B 16.1506,C -0.105,E1 16.1528,E2 539.0156} C_DIS
Enddeposition()
LIN {X 0.9586,Y -136.2769,Z 156,A -92.8363,B 24.9708,C -1.2495,E1 25.0007,E2 539.5159} C_DIS
Startdeposition()
$VEL.CP = VEL_PRINT
LIN {X 4.8365,Y -136.1962,Z 156,A -90.5835,B 24.9691,C -1.2838,E1 25.0072,E2 537.1824} C_DIS
LIN {X 8.6611,Y -136.006,Z 156,A -88.9239,B 24.969,C -1.2872,E1 25.0118,E2 535.5153} C_DIS
LIN {X 13.3133,Y -135.6296,Z 156,A -87.0224,B 24.969,C -1.2849,E1 25.0171,E2 533.6204} C_DIS
LIN {X 17.0691,Y -135.2095,Z 156,A -85.3372,B 24.9688,C -1.2912,E1 25.0218,E2 531.9217} C_DIS
LIN {X 21.2838,Y -134.6095,Z 156,A -83.6929,B 24.9691,C -1.2845,E1 25.0263,E2 530.2948} C_DIS
LIN {X 24.796,Y -134.0086,Z 156,A -82.1315,B 24.9689,C -1.2891,E1 25.0306,E2 528.7239} C_DIS
LIN {X 28.2522,Y -133.3214,Z 156,A -80.5876,B 24.9686,C -1.294,E1 25.0349,E2 527.1706} C_DIS
LIN {X 32.3613,Y -132.3837,Z 156,A -78.9097,B 24.9688,C -1.2905,E1 25.0394,E2 525.5032} C_DIS
LIN {X 35.9736,Y -131.4495,Z 156,A -77.3287,B 24.9687,C -1.2929,E1 25.0437,E2 523.9191} C_DIS
LIN {X 39.3245,Y -130.4853,Z 156,A -75.9519,B 24.9689,C -1.2896,E1 25.0473,E2 522.5524} C_DIS
LIN {X 42.6247,Y -129.4442,Z 156,A -74.3536,B 24.9684,C -1.2994,E1 25.0516,E2 520.9339} C_DIS
LIN {X 46.522,Y -128.0948,Z 156,A -72.7192,B 24.9685,C -1.2962,E1 25.0559,E2 519.3105} C_DIS
LIN {X 50.5633,Y -126.5542,Z 156,A -70.8864,B 24.9684,C -1.2996,E1 25.0607,E2 517.4737} C_DIS
LIN {X 53.8191,Y -125.204,Z 156,A -69.4146,B 24.9683,C -1.3013,E1 25.0645,E2 516.0014} C_DIS
LIN {X 57.403,Y -123.6017,Z 156,A -67.7518,B 24.9681,C -1.3046,E1 25.0687,E2 514.3349} C_DIS
LIN {X 60.9802,Y -121.8788,Z 156,A -65.9902,B 24.9677,C -1.3125,E1 25.0731,E2 512.5593} C_DIS
LIN {X 64.8063,Y -119.8884,Z 156,A -64.2658,B 24.9678,C -1.3107,E1 25.0774,E2 510.844} C_DIS
LIN {X 68.6302,Y -117.7414,Z 156,A -62.4648,B 24.9678,C -1.3117,E1 25.0817,E2 509.046} C_DIS
LIN {X 71.8519,Y -115.8028,Z 156,A -60.8264,B 24.9675,C -1.318,E1 25.0857,E2 507.398} C_DIS
LIN {X 75.3772,Y -113.5401,Z 156,A -59.0572,B 24.9673,C -1.322,E1 25.0898,E2 505.6251} C_DIS
LIN {X 79.0339,Y -111.0256,Z 156,A -57.1908,B 24.9671,C -1.326,E1 25.0941,E2 503.7558} C_DIS
LIN {X 82.5083,Y -108.4688,Z 156,A -55.3914,B 24.9669,C -1.3291,E1 25.0981,E2 501.9555} C_DIS
LIN {X 86.0128,Y -105.7112,Z 156,A -53.5207,B 24.9667,C -1.3331,E1 25.1022,E2 500.0824} C_DIS
LIN {X 89.5633,Y -102.7199,Z 156,A -51.6249,B 24.9667,C -1.3345,E1 25.1062,E2 498.1908} C_DIS
LIN {X 92.4367,Y -100.1424,Z 156,A -50.0642,B 24.9667,C -1.3348,E1 25.1094,E2 496.6355} C_DIS
LIN {X 94.9918,Y -97.7221,Z 156,A -48.531,B 24.9663,C -1.3415,E1 25.1125,E2 495.0929} C_DIS
LIN {X 97.8153,Y -94.8954,Z 156,A -46.8647,B 24.9661,C -1.345,E1 25.1158,E2 493.4255} C_DIS
LIN {X 100.8718,Y -91.6398,Z 156,A -44.9993,B 24.9659,C -1.3492,E1 25.1193,E2 491.5583} C_DIS
LIN {X 103.8474,Y -88.2535,Z 156,A -43.1243,B 24.9657,C -1.3531,E1 25.1227,E2 489.6827} C_DIS
LIN {X 106.6775,Y -84.8108,Z 156,A -41.3017,B 24.9656,C -1.3553,E1 25.1259,E2 487.8634} C_DIS
LIN {X 108.9121,Y -81.9217,Z 156,A -39.6897,B 24.9652,C -1.3639,E1 25.1287,E2 486.2387} C_DIS
LIN {X 111.3751,Y -78.5401,Z 156,A -38.0272,B 24.9652,C -1.3634,E1 25.1314,E2 484.5855} C_DIS
LIN {X 113.7298,Y -75.0901,Z 156,A -36.2769,B 24.9649,C -1.3681,E1 25.1341,E2 482.8328} C_DIS
LIN {X 115.75,Y -71.9369,Z 156,A -34.6368,B 24.9645,C -1.3765,E1 25.1365,E2 481.1812} C_DIS
LIN {X 118.1612,Y -67.905,Z 156,A -32.6554,B 24.9642,C -1.3827,E1 25.1393,E2 479.1953} C_DIS
LIN {X 120.1742,Y -64.2744,Z 156,A -30.8992,B 24.9639,C -1.3887,E1 25.1417,E2 477.4344} C_DIS
LIN {X 122.1036,Y -60.5245,Z 156,A -29.2476,B 24.9639,C -1.3871,E1 25.1438,E2 475.7951} C_DIS
LIN {X 123.6263,Y -57.3498,Z 156,A -27.8329,B 24.9639,C -1.388,E1 25.1454,E2 474.3861} C_DIS
LIN {X 124.864,Y -54.6054,Z 156,A -26.5816,B 24.9638,C -1.3911,E1 25.1468,E2 473.1343} C_DIS
LIN {X 126.2275,Y -51.3738,Z 156,A -24.9735,B 24.9631,C -1.4034,E1 25.1486,E2 471.5059} C_DIS
LIN {X 127.7057,Y -47.579,Z 156,A -23.3861,B 24.9631,C -1.4017,E1 25.1501,E2 469.9315} C_DIS
LIN {X 129.0319,Y -43.8625,Z 156,A -21.6457,B 24.9627,C -1.4117,E1 25.1518,E2 468.1774} C_DIS
LIN {X 130.2364,Y -40.1377,Z 156,A -20.1253,B 24.9627,C -1.4098,E1 25.153,E2 466.67} C_DIS
LIN {X 131.1614,Y -37.0038,Z 156,A -18.7042,B 24.9624,C -1.417,E1 25.1541,E2 465.2401} C_DIS
LIN {X 132.1241,Y -33.4025,Z 156,A -17.1967,B 24.9623,C -1.4187,E1 25.1552,E2 463.7373} C_DIS
LIN {X 132.8947,Y -30.1917,Z 156,A -15.8243,B 24.9621,C -1.4223,E1 25.1561,E2 462.3642} C_DIS
LIN {X 133.6303,Y -26.7514,Z 156,A -14.2169,B 24.9614,C -1.4346,E1 25.157,E2 460.7373} C_DIS
LIN {X 134.401,Y -22.5594,Z 156,A -12.5657,B 24.9616,C -1.4324,E1 25.1578,E2 459.101} C_DIS
LIN {X 134.9094,Y -19.2872,Z 156,A -11.1538,B 24.9613,C -1.4381,E1 25.1583,E2 457.6839} C_DIS
LIN {X 135.3935,Y -15.5406,Z 156,A -9.6243,B 24.9612,C -1.44,E1 25.1589,E2 456.159} C_DIS
LIN {X 135.75,Y -12.0339,Z 156,A -8.1164,B 24.9608,C -1.4464,E1 25.1593,E2 454.6448} C_DIS
LIN {X 136.0375,Y -8.1501,Z 156,A -6.4874,B 24.9605,C -1.4514,E1 25.1596,E2 453.0137} C_DIS
LIN {X 136.216,Y -4.2404,Z 156,A -4.8727,B 24.9603,C -1.4551,E1 25.1597,E2 451.4} C_DIS
LIN {X 136.2783,Y -0.9663,Z 156,A -3.4658,B 24.96,C -1.4614,E1 25.1597,E2 449.9866} C_DIS
LIN {X 136.2449,Y 3.203,Z 156,A -1.6757,B 24.9596,C -1.4694,E1 25.1597,E2 448.1884} C_DIS
LIN {X 136.0968,Y 7.0918,Z 156,A -0.0396,B 24.9593,C -1.4748,E1 25.1595,E2 446.5492} C_DIS
LIN {X 135.8119,Y 11.3011,Z 156,A 1.6148,B 24.9593,C -1.4738,E1 25.1592,E2 444.907} C_DIS
LIN {X 135.5012,Y 14.5591,Z 156,A 3.0258,B 24.9589,C -1.4803,E1 25.1587,E2 443.4891} C_DIS
LIN {X 135.0385,Y 18.3736,Z 156,A 4.5756,B 24.9589,C -1.4818,E1 25.1582,E2 441.9449} C_DIS
LIN {X 134.5178,Y 21.8591,Z 156,A 6.0594,B 24.9586,C -1.4867,E1 25.1576,E2 440.4582} C_DIS
LIN {X 133.9068,Y 25.3291,Z 156,A 7.5797,B 24.9582,C -1.4938,E1 25.1568,E2 438.9303} C_DIS
LIN {X 133.2405,Y 28.627,Z 156,A 8.9311,B 24.9582,C -1.4947,E1 25.156,E2 437.5846} C_DIS
LIN {X 132.5173,Y 31.8068,Z 156,A 10.2119,B 24.9582,C -1.4939,E1 25.1552,E2 436.313} C_DIS
LIN {X 131.6538,Y 35.2105,Z 156,A 11.7957,B 24.9576,C -1.5047,E1 25.1541,E2 434.7129} C_DIS
LIN {X 130.606,Y 38.9228,Z 156,A 13.5171,B 24.957,C -1.5155,E1 25.1527,E2 432.9759} C_DIS
LIN {X 129.3573,Y 42.8857,Z 156,A 15.0992,B 24.9572,C -1.5115,E1 25.1514,E2 431.4122} C_DIS
LIN {X 128.2227,Y 46.1672,Z 156,A 16.5721,B 24.9569,C -1.5167,E1 25.15,E2 429.9353} C_DIS
LIN {X 127.0294,Y 49.3557,Z 156,A 17.9788,B 24.9567,C -1.5196,E1 25.1486,E2 428.5296} C_DIS
LIN {X 125.9768,Y 51.9868,Z 156,A 19.1541,B 24.9566,C -1.5222,E1 25.1474,E2 427.3545} C_DIS
LIN {X 124.5904,Y 55.2257,Z 156,A 20.6288,B 24.9564,C -1.5262,E1 25.1457,E2 425.8785} C_DIS
LIN {X 123.1569,Y 58.3523,Z 156,A 22.1277,B 24.9559,C -1.5335,E1 25.144,E2 424.3706} C_DIS
LIN {X 121.623,Y 61.4852,Z 156,A 23.5815,B 24.9557,C -1.537,E1 25.1421,E2 422.9163} C_DIS
LIN {X 120.0177,Y 64.5657,Z 156,A 25.1005,B 24.9553,C -1.5444,E1 25.1401,E2 421.3877} C_DIS
LIN {X 117.9929,Y 68.1957,Z 156,A 26.7814,B 24.9553,C -1.5455,E1 25.1378,E2 419.7131} C_DIS
LIN {X 115.7837,Y 71.8826,Z 156,A 28.5654,B 24.955,C -1.5491,E1 25.1352,E2 417.9296} C_DIS
LIN {X 113.883,Y 74.8575,Z 156,A 30.1081,B 24.9546,C -1.5564,E1 25.1329,E2 416.3774} C_DIS
LIN {X 111.371,Y 78.5459,Z 156,A 31.9428,B 24.9545,C -1.5589,E1 25.13,E2 414.5458} C_DIS
LIN {X 108.6744,Y 82.2367,Z 156,A 33.9042,B 24.954,C -1.566,E1 25.1267,E2 412.5769} C_DIS
LIN {X 106.066,Y 85.5743,Z 156,A 35.5851,B 24.9541,C -1.5648,E1 25.1238,E2 410.9069} C_DIS
LIN {X 103.3785,Y 88.8025,Z 156,A 37.3474,B 24.9539,C -1.5688,E1 25.1206,E2 409.1431} C_DIS
LIN {X 100.5921,Y 91.9475,Z 156,A 39.1724,B 24.9534,C -1.5762,E1 25.1172,E2 407.3088} C_DIS
LIN {X 97.9663,Y 94.7395,Z 156,A 40.7777,B 24.9533,C -1.5795,E1 25.1141,E2 405.7027} C_DIS
LIN {X 94.9328,Y 97.7791,Z 156,A 42.5068,B 24.9533,C -1.5792,E1 25.1106,E2 403.9816} C_DIS
LIN {X 91.8806,Y 100.6533,Z 156,A 44.2693,B 24.9531,C -1.5829,E1 25.107,E2 402.2175} C_DIS
LIN {X 89.0567,Y 103.1596,Z 156,A 45.9102,B 24.9527,C -1.5891,E1 25.1036,E2 400.5685} C_DIS
LIN {X 85.4465,Y 106.1691,Z 156,A 47.7869,B 24.9527,C -1.5874,E1 25.0995,E2 398.7029} C_DIS
LIN {X 82.3772,Y 108.5683,Z 156,A 49.4322,B 24.9526,C -1.5909,E1 25.0959,E2 397.0554} C_DIS
LIN {X 79.0344,Y 111.0252,Z 156,A 51.2283,B 24.9522,C -1.5969,E1 25.0918,E2 395.2515} C_DIS
LIN {X 75.3492,Y 113.5588,Z 156,A 53.0824,B 24.9522,C -1.5986,E1 25.0875,E2 393.3996} C_DIS
LIN {X 71.7986,Y 115.836,Z 156,A 54.8323,B 24.952,C -1.6001,E1 25.0834,E2 391.6516} C_DIS
LIN {X 68.4793,Y 117.8287,Z 156,A 56.5126,B 24.9517,C -1.6055,E1 25.0793,E2 389.9638} C_DIS
LIN {X 64.8459,Y 119.8672,Z 156,A 58.2813,B 24.9515,C -1.6089,E1 25.075,E2 388.1921} C_DIS
LIN {X 60.8278,Y 121.954,Z 156,A 60.0261,B 24.9519,C -1.6027,E1 25.0707,E2 386.4667} C_DIS
LIN {X 57.6541,Y 123.4856,Z 156,A 61.5089,B 24.9518,C -1.6047,E1 25.067,E2 384.9833} C_DIS
LIN {X 54.6721,Y 124.8351,Z 156,A 62.9562,B 24.9514,C -1.6102,E1 25.0633,E2 383.5265} C_DIS
LIN {X 51.4196,Y 126.2091,Z 156,A 64.4315,B 24.9514,C -1.6113,E1 25.0594,E2 382.052} C_DIS
LIN {X 48.1418,Y 127.4949,Z 156,A 65.8794,B 24.9514,C -1.611,E1 25.0557,E2 380.6079} C_DIS
LIN {X 44.7151,Y 128.7363,Z 156,A 67.3711,B 24.9514,C -1.6102,E1 25.0518,E2 379.1211} C_DIS
LIN {X 41.6516,Y 129.76,Z 156,A 68.7401,B 24.9514,C -1.612,E1 25.0481,E2 377.7505} C_DIS
LIN {X 38.9111,Y 130.6094,Z 156,A 69.9321,B 24.9514,C -1.612,E1 25.045,E2 376.5604} C_DIS
LIN {X 35.7739,Y 131.5036,Z 156,A 71.3785,B 24.951,C -1.6171,E1 25.041,E2 375.1045} C_DIS
LIN {X 32.3726,Y 132.381,Z 156,A 72.8597,B 24.951,C -1.6183,E1 25.037,E2 373.6227} C_DIS
LIN {X 28.1896,Y 133.3349,Z 156,A 74.6051,B 24.951,C -1.616,E1 25.0323,E2 371.8849} C_DIS
LIN {X 24.7327,Y 134.02,Z 156,A 76.1447,B 24.9508,C -1.6198,E1 25.028,E2 370.3383} C_DIS
LIN {X 21.2588,Y 134.6134,Z 156,A 77.6058,B 24.9508,C -1.6192,E1 25.024,E2 368.88} C_DIS
LIN {X 17.0241,Y 135.2154,Z 156,A 79.4034,B 24.9508,C -1.6196,E1 25.019,E2 367.0829} C_DIS
LIN {X 13.2607,Y 135.6347,Z 156,A 81.0428,B 24.9507,C -1.6224,E1 25.0145,E2 365.438} C_DIS
LIN {X 8.9095,Y 135.9907,Z 156,A 82.8916,B 24.9507,C -1.6232,E1 25.0093,E2 363.5882} C_DIS
LIN {X 4.5963,Y 136.2056,Z 156,A 84.598,B 24.951,C -1.6172,E1 25.0046,E2 361.8964} C_DIS
LIN {X 0.5681,Y 136.2803,Z 156,A 86.2973,B 24.951,C -1.6172,E1 24.9999,E2 360.1972} C_DIS
LIN {X -3.2121,Y 136.2446,Z 156,A 87.884,B 24.951,C -1.6167,E1 24.9954,E2 358.6117} C_DIS
LIN {X -6.7375,Y 136.1146,Z 156,A 89.446,B 24.9508,C -1.6204,E1 24.991,E2 357.0406} C_DIS
LIN {X -11.0153,Y 135.8361,Z 156,A 91.2425,B 24.9508,C -1.6193,E1 24.986,E2 355.246} C_DIS
LIN {X -15.2113,Y 135.431,Z 156,A 92.98,B 24.951,C -1.6165,E1 24.9812,E2 353.5142} C_DIS
LIN {X -18.7097,Y 134.9919,Z 156,A 94.4876,B 24.951,C -1.6169,E1 24.9771,E2 352.0044} C_DIS
LIN {X -22.1913,Y 134.4624,Z 156,A 95.9104,B 24.9513,C -1.6128,E1 24.9732,E2 350.59} C_DIS
LIN {X -25.4529,Y 133.8831,Z 156,A 97.1896,B 24.9517,C -1.6058,E1 24.9697,E2 349.3263} C_DIS
LIN {X -28.2864,Y 133.314,Z 156,A 98.6545,B 24.951,C -1.6178,E1 24.9656,E2 347.8311} C_DIS
LIN {X -32.3829,Y 132.3785,Z 156,A 100.2991,B 24.9514,C -1.6097,E1 24.9612,E2 346.2034} C_DIS
LIN {X -35.782,Y 131.5014,Z 156,A 101.8021,B 24.9514,C -1.6096,E1 24.9571,E2 344.6984} C_DIS
LIN {X -39.1586,Y 130.536,Z 156,A 103.2337,B 24.9517,C -1.6056,E1 24.9533,E2 343.274} C_DIS
LIN {X -42.5104,Y 129.4823,Z 156,A 104.7147,B 24.9517,C -1.604,E1 24.9494,E2 341.794} C_DIS
LIN {X -45.9258,Y 128.3097,Z 156,A 106.2632,B 24.9518,C -1.6037,E1 24.9453,E2 340.2433} C_DIS
LIN {X -49.075,Y 127.1385,Z 156,A 107.7158,B 24.9518,C -1.6038,E1 24.9415,E2 338.7874} C_DIS
LIN {X -52.9757,Y 125.5638,Z 156,A 109.4592,B 24.952,C -1.6,E1 24.937,E2 337.0491} C_DIS
LIN {X -56.4273,Y 124.0528,Z 156,A 111.0342,B 24.9522,C -1.597,E1 24.933,E2 335.4773} C_DIS
LIN {X -59.9978,Y 122.3634,Z 156,A 112.5115,B 24.9529,C -1.585,E1 24.9293,E2 334.025} C_DIS
LIN {X -62.5229,Y 121.0947,Z 156,A 114.0187,B 24.9521,C -1.5994,E1 24.9255,E2 332.4794} C_DIS
LIN {X -66.5269,Y 118.9421,Z 156,A 115.9291,B 24.9523,C -1.596,E1 24.9208,E2 330.5717} C_DIS
LIN {X -70.0586,Y 116.8968,Z 156,A 117.6677,B 24.9523,C -1.5939,E1 24.9166,E2 328.8326} C_DIS
LIN {X -73.6508,Y 114.6672,Z 156,A 119.414,B 24.9527,C -1.5889,E1 24.9125,E2 327.0928} C_DIS
LIN {X -77.4087,Y 112.165,Z 156,A 121.3285,B 24.9529,C -1.5859,E1 24.9081,E2 325.1789} C_DIS
LIN {X -80.5232,Y 109.9501,Z 156,A 122.947,B 24.953,C -1.5831,E1 24.9044,E2 323.5614} C_DIS
LIN {X -83.8574,Y 107.4294,Z 156,A 124.6444,B 24.9534,C -1.5762,E1 24.9007,E2 321.8743} C_DIS
LIN {X -87.0999,Y 104.8171,Z 156,A 126.3887,B 24.9537,C -1.572,E1 24.8969,E2 320.1335} C_DIS
LIN {X -90.2084,Y 102.1539,Z 156,A 128.1672,B 24.9537,C -1.5709,E1 24.8932,E2 318.3504} C_DIS
LIN {X -93.1713,Y 99.4597,Z 156,A 129.8204,B 24.9541,C -1.5653,E1 24.8898,E2 316.7039} C_DIS
LIN {X -96.1751,Y 96.5574,Z 156,A 131.5809,B 24.9543,C -1.5613,E1 24.8863,E2 314.9457} C_DIS
LIN {X -99.0849,Y 93.569,Z 156,A 133.3856,B 24.9544,C -1.5594,E1 24.8828,E2 313.1376} C_DIS
LIN {X -101.7781,Y 90.633,Z 156,A 135.1219,B 24.9545,C -1.5582,E1 24.8796,E2 311.3965} C_DIS
LIN {X -104.6438,Y 87.3086,Z 156,A 136.9751,B 24.9548,C -1.5537,E1 24.8762,E2 309.5455} C_DIS
LIN {X -107.2436,Y 84.0939,Z 156,A 138.7081,B 24.9551,C -1.5487,E1 24.8732,E2 307.8163} C_DIS
LIN {X -109.7495,Y 80.7962,Z 156,A 140.3868,B 24.9555,C -1.5407,E1 24.8704,E2 306.1486} C_DIS
LIN {X -111.8947,Y 77.7982,Z 156,A 142.0391,B 24.9555,C -1.5415,E1 24.8678,E2 304.4862} C_DIS
LIN {X -114.4192,Y 74.0355,Z 156,A 143.9506,B 24.9558,C -1.5364,E1 24.8648,E2 302.5774} C_DIS
LIN {X -116.6556,Y 70.4589,Z 156,A 145.6454,B 24.9563,C -1.5272,E1 24.8624,E2 300.8957} C_DIS
LIN {X -118.7795,Y 66.8162,Z 156,A 147.4525,B 24.9565,C -1.5237,E1 24.8599,E2 299.0877} C_DIS
LIN {X -120.5264,Y 63.6074,Z 156,A 148.9831,B 24.9568,C -1.5188,E1 24.8578,E2 297.5605} C_DIS
LIN {X -122.1211,Y 60.489,Z 156,A 150.4625,B 24.957,C -1.5146,E1 24.856,E2 296.083} C_DIS
LIN {X -123.6324,Y 57.3366,Z 156,A 151.8862,B 24.9574,C -1.5078,E1 24.8543,E2 294.6679} C_DIS
LIN {X -125.0616,Y 54.1484,Z 156,A 153.3668,B 24.9576,C -1.5038,E1 24.8526,E2 293.1887} C_DIS
LIN {X -126.3157,Y 51.155,Z 156,A 154.7649,B 24.9578,C -1.5012,E1 24.8512,E2 291.7889} C_DIS
LIN {X -127.3883,Y 48.4264,Z 156,A 155.9784,B 24.9581,C -1.4963,E1 24.8499,E2 290.5803} C_DIS
LIN {X -128.5151,Y 45.353,Z 156,A 157.4982,B 24.9579,C -1.4991,E1 24.8485,E2 289.0452} C_DIS
LIN {X -129.7029,Y 41.8302,Z 156,A 159.0004,B 24.9583,C -1.4911,E1 24.8472,E2 287.5535} C_DIS
LIN {X -130.9213,Y 37.846,Z 156,A 160.7266,B 24.9587,C -1.4842,E1 24.8458,E2 285.8339} C_DIS
LIN {X -132.0116,Y 33.8459,Z 156,A 162.2941,B 24.9595,C -1.4697,E1 24.8447,E2 284.2918} C_DIS
LIN {X -132.7468,Y 30.839,Z 156,A 163.7849,B 24.9592,C -1.4749,E1 24.8437,E2 282.7798} C_DIS
LIN {X -133.4535,Y 27.6204,Z 156,A 165.1677,B 24.9595,C -1.4702,E1 24.8429,E2 281.4} C_DIS
LIN {X -134.1313,Y 24.1108,Z 156,A 166.6816,B 24.9597,C -1.4659,E1 24.8421,E2 279.8876} C_DIS
LIN {X -134.6689,Y 20.9003,Z 156,A 168.1009,B 24.9599,C -1.4639,E1 24.8415,E2 278.4646} C_DIS
LIN {X -135.1624,Y 17.4282,Z 156,A 169.5655,B 24.9601,C -1.4585,E1 24.841,E2 277.004} C_DIS
LIN {X -135.5781,Y 13.8447,Z 156,A 171.1498,B 24.9602,C -1.4568,E1 24.8405,E2 275.4142} C_DIS
LIN {X -135.8893,Y 10.3361,Z 156,A 172.5715,B 24.9607,C -1.449,E1 24.8402,E2 274.0027} C_DIS
LIN {X -136.1103,Y 6.8236,Z 156,A 174.0521,B 24.9609,C -1.4441,E1 24.8399,E2 272.5247} C_DIS
LIN {X -136.2421,Y 3.3046,Z 156,A 175.6827,B 24.9608,C -1.4467,E1 24.8399,E2 270.8781} C_DIS
LIN {X -136.2797,Y -0.6754,Z 156,A 177.2803,B 24.9613,C -1.4374,E1 24.8398,E2 269.293} C_DIS
LIN {X -136.2084,Y -4.5168,Z 156,A 178.8642,B 24.9617,C -1.4305,E1 24.8399,E2 267.7162} C_DIS
LIN {X -136.0449,Y -8.03,Z 156,A -179.6479,B 24.9619,C -1.4261,E1 24.8401,E2 266.2298} C_DIS
LIN {X -135.8133,Y -11.2849,Z 156,A -178.2471,B 24.9621,C -1.423,E1 24.8404,E2 264.8278} C_DIS
LIN {X -135.4648,Y -14.8973,Z 156,A -176.7185,B 24.9623,C -1.4182,E1 24.8409,E2 263.3017} C_DIS
LIN {X -135.0379,Y -18.3786,Z 156,A -175.2587,B 24.9626,C -1.4126,E1 24.8414,E2 261.8463} C_DIS
LIN {X -134.5195,Y -21.8491,Z 156,A -173.7628,B 24.9628,C -1.4089,E1 24.842,E2 260.3505} C_DIS
LIN {X -133.8671,Y -25.5366,Z 156,A -172.1826,B 24.9631,C -1.4041,E1 24.8428,E2 258.7722} C_DIS
LIN {X -133.2237,Y -28.7047,Z 156,A -170.8172,B 24.9633,C -1.4001,E1 24.8436,E2 257.4084} C_DIS
LIN {X -132.511,Y -31.8331,Z 156,A -169.5068,B 24.9636,C -1.3939,E1 24.8444,E2 256.1051} C_DIS
LIN {X -131.6634,Y -35.1746,Z 156,A -167.9611,B 24.9636,C -1.3942,E1 24.8455,E2 254.5498} C_DIS
LIN {X -130.6224,Y -38.8669,Z 156,A -166.2242,B 24.9636,C -1.3954,E1 24.8469,E2 252.7999} C_DIS
LIN {X -129.355,Y -42.8926,Z 156,A -164.5861,B 24.9642,C -1.383,E1 24.8483,E2 251.1818} C_DIS
LIN {X -128.2614,Y -46.0597,Z 156,A -163.315,B 24.9648,C -1.3718,E1 24.8494,E2 249.9303} C_DIS
LIN {X -127.1625,Y -49.0132,Z 156,A -161.9599,B 24.9648,C -1.3693,E1 24.8508,E2 248.5735} C_DIS
LIN {X -125.9807,Y -51.9775,Z 156,A -160.4933,B 24.9648,C -1.3716,E1 24.8523,E2 247.0932} C_DIS
LIN {X -124.5973,Y -55.2103,Z 156,A -159.0056,B 24.965,C -1.3677,E1 24.854,E2 245.6066} C_DIS
LIN {X -123.2393,Y -58.1799,Z 156,A -157.5496,B 24.965,C -1.3679,E1 24.8557,E2 244.1421} C_DIS
LIN {X -121.6958,Y -61.3421,Z 156,A -156.0459,B 24.9651,C -1.3649,E1 24.8576,E2 242.6375} C_DIS
LIN {X -120.0077,Y -64.5844,Z 156,A -154.453,B 24.9651,C -1.3634,E1 24.8597,E2 241.0397} C_DIS
LIN {X -117.9535,Y -68.2638,Z 156,A -152.7538,B 24.9656,C -1.3548,E1 24.862,E2 239.3521} C_DIS
LIN {X -115.7909,Y -71.8712,Z 156,A -150.9704,B 24.9658,C -1.3508,E1 24.8646,E2 237.5691} C_DIS
LIN {X -113.7563,Y -75.0499,Z 156,A -149.2964,B 24.9658,C -1.3511,E1 24.8672,E2 235.8861} C_DIS
LIN {X -111.3499,Y -78.5759,Z 156,A -147.5705,B 24.9662,C -1.3429,E1 24.8699,E2 234.1712} C_DIS
LIN {X -109.2097,Y -81.5244,Z 156,A -145.9531,B 24.9662,C -1.3434,E1 24.8726,E2 232.5447} C_DIS
LIN {X -106.656,Y -84.8378,Z 156,A -144.1825,B 24.9664,C -1.3397,E1 24.8757,E2 230.7746} C_DIS
LIN {X -103.8456,Y -88.2556,Z 156,A -142.3829,B 24.9668,C -1.3321,E1 24.8789,E2 228.9849} C_DIS
LIN {X -101.0294,Y -91.4661,Z 156,A -140.5877,B 24.967,C -1.3279,E1 24.8822,E2 227.1916} C_DIS
LIN {X -98.15,Y -94.5498,Z 156,A -138.7794,B 24.967,C -1.3257,E1 24.8857,E2 225.3807} C_DIS
LIN {X -95.4278,Y -97.296,Z 156,A -137.2261,B 24.9674,C -1.3184,E1 24.8887,E2 223.8381} C_DIS
LIN {X -92.8967,Y -99.7154,Z 156,A -135.7487,B 24.9676,C -1.3156,E1 24.8917,E2 222.3614} C_DIS
LIN {X -89.9794,Y -102.3563,Z 156,A -134.0375,B 24.9676,C -1.3151,E1 24.8953,E2 220.6444} C_DIS
LIN {X -87.1277,Y -104.7941,Z 156,A -132.3609,B 24.9676,C -1.3172,E1 24.8989,E2 218.9565} C_DIS
LIN {X -83.7376,Y -107.5224,Z 156,A -130.6064,B 24.9679,C -1.3099,E1 24.9027,E2 217.2129} C_DIS
LIN {X -80.3705,Y -110.0623,Z 156,A -128.8307,B 24.968,C -1.3068,E1 24.9067,E2 215.4381} C_DIS
LIN {X -77.2866,Y -112.2488,Z 156,A -127.1648,B 24.968,C -1.3081,E1 24.9105,E2 213.7635} C_DIS
LIN {X -73.7805,Y -114.5842,Z 156,A -125.4788,B 24.9683,C -1.3008,E1 24.9144,E2 212.0894} C_DIS
LIN {X -70.6935,Y -116.5137,Z 156,A -123.8585,B 24.9682,C -1.3031,E1 24.9183,E2 210.4585} C_DIS
LIN {X -67.126,Y -118.6054,Z 156,A -122.1575,B 24.9684,C -1.2986,E1 24.9224,E2 208.7632} C_DIS
LIN {X -63.9761,Y -120.3328,Z 156,A -120.7299,B 24.9687,C -1.2922,E1 24.9259,E2 207.3468} C_DIS
LIN {X -60.8424,Y -121.9468,Z 156,A -119.1099,B 24.9685,C -1.2976,E1 24.93,E2 205.7096} C_DIS
LIN {X -57.6677,Y -123.4793,Z 156,A -117.7517,B 24.9689,C -1.2892,E1 24.9334,E2 204.3678} C_DIS
LIN {X -54.6866,Y -124.8289,Z 156,A -116.2957,B 24.9687,C -1.2919,E1 24.9371,E2 202.902} C_DIS
LIN {X -51.4372,Y -126.202,Z 156,A -114.7822,B 24.9687,C -1.2919,E1 24.941,E2 201.3849} C_DIS
LIN {X -48.0413,Y -127.5326,Z 156,A -113.3492,B 24.9691,C -1.2851,E1 24.9447,E2 199.965} C_DIS
LIN {X -44.7689,Y -128.7176,Z 156,A -111.8677,B 24.9691,C -1.2848,E1 24.9486,E2 198.4814} C_DIS
LIN {X -41.6333,Y -129.7658,Z 156,A -110.485,B 24.9691,C -1.2833,E1 24.9523,E2 197.0997} C_DIS
LIN {X -38.9365,Y -130.602,Z 156,A -109.2979,B 24.9691,C -1.2824,E1 24.9555,E2 195.9128} C_DIS
LIN {X -35.7991,Y -131.4968,Z 156,A -107.8269,B 24.969,C -1.2868,E1 24.9595,E2 194.4291} C_DIS
LIN {X -32.3185,Y -132.394,Z 156,A -106.3459,B 24.9691,C -1.2843,E1 24.9635,E2 192.9518} C_DIS
LIN {X -28.207,Y -133.3312,Z 156,A -104.6141,B 24.9693,C -1.2812,E1 24.9682,E2 191.2251} C_DIS
LIN {X -24.7493,Y -134.017,Z 156,A -103.0668,B 24.9691,C -1.2842,E1 24.9724,E2 189.6692} C_DIS
LIN {X -21.2748,Y -134.6109,Z 156,A -101.6464,B 24.9693,C -1.2804,E1 24.9763,E2 188.2565} C_DIS
LIN {X -17.7243,Y -135.1236,Z 156,A -100.1571,B 24.9693,C -1.2791,E1 24.9805,E2 186.7691} C_DIS
LIN {X -14.2216,Y -135.5375,Z 156,A -98.5497,B 24.969,C -1.2856,E1 24.985,E2 185.1452} C_DIS
LIN {X -10.0185,Y -135.9125,Z 156,A -96.8571,B 24.9693,C -1.2811,E1 24.9896,E2 183.4625} C_DIS
LIN {X -6.496,Y -136.1268,Z 156,A -95.4011,B 24.9693,C -1.2797,E1 24.9937,E2 182.0095} C_DIS
LIN {X -2.9146,Y -136.2517,Z 156,A -93.7488,B 24.9689,C -1.2878,E1 24.9984,E2 180.3378} C_DIS
LIN {X 0.9586,Y -136.2769,Z 156,A -92.8359,B 24.9708,C -1.2494,E1 25.0007,E2 179.5159} C_DIS
Enddeposition()
LIN {X 0.9586,Y -136.2769,Z 156,A -92.8359,B 24.9708,C -1.2494,E1 25.0007,E2 179.5159} C_DIS
Startdeposition()
$VEL.CP = VEL_PRINT
LIN {X -1.0918,Y -135.3436,Z 156,A -93.8189,B 24.9703,C -1.2595,E1 24.998,E2 180.475} C_DIS
LIN {X -5.0736,Y -135.2525,Z 156,A -95.5109,B 24.9703,C -1.2589,E1 24.9933,E2 182.1686} C_DIS
LIN {X -8.7972,Y -135.0621,Z 156,A -97.1715,B 24.9705,C -1.2545,E1 24.9886,E2 183.8402} C_DIS
LIN {X -12.851,Y -134.736,Z 156,A -98.7969,B 24.9703,C -1.2597,E1 24.9841,E2 185.4539} C_DIS
LIN {X -16.3358,Y -134.3583,Z 156,A -100.3465,B 24.9704,C -1.2564,E1 24.9798,E2 187.0123} C_DIS
LIN {X -20.715,Y -133.7527,Z 156,A -102.1526,B 24.9702,C -1.2604,E1 24.9748,E2 188.8106} C_DIS
LIN {X -24.3075,Y -133.1475,Z 156,A -103.7891,B 24.9705,C -1.2559,E1 24.9703,E2 190.4593} C_DIS
LIN {X -28.454,Y -132.3225,Z 156,A -105.5164,B 24.9703,C -1.26,E1 24.9656,E2 192.1789} C_DIS
LIN {X -31.8624,Y -131.5434,Z 156,A -106.9557,B 24.9701,C -1.2629,E1 24.9617,E2 193.6133} C_DIS
LIN {X -35.0104,Y -130.7408,Z 156,A -108.3183,B 24.9701,C -1.2644,E1 24.958,E2 194.9743} C_DIS
LIN {X -38.1264,Y -129.8662,Z 156,A -109.7234,B 24.9701,C -1.2635,E1 24.9542,E2 196.3837} C_DIS
LIN {X -41.4706,Y -128.8376,Z 156,A -111.2216,B 24.9701,C -1.2638,E1 24.9502,E2 197.8839} C_DIS
LIN {X -44.5916,Y -127.7908,Z 156,A -112.632,B 24.9701,C -1.2641,E1 24.9465,E2 199.2964} C_DIS
LIN {X -48.9091,Y -126.2012,Z 156,A -114.6027,B 24.9701,C -1.2648,E1 24.9413,E2 201.2695} C_DIS
LIN {X -52.3126,Y -124.8288,Z 156,A -116.1123,B 24.9699,C -1.2687,E1 24.9374,E2 202.7732} C_DIS
LIN {X -55.6313,Y -123.3861,Z 156,A -117.6074,B 24.9697,C -1.2723,E1 24.9336,E2 204.2634} C_DIS
LIN {X -58.6194,Y -121.9945,Z 156,A -119.0308,B 24.9697,C -1.2725,E1 24.93,E2 205.6897} C_DIS
LIN {X -61.7005,Y -120.4656,Z 156,A -120.4913,B 24.9696,C -1.2742,E1 24.9264,E2 207.1503} C_DIS
LIN {X -64.6697,Y -118.8999,Z 156,A -122.0406,B 24.9698,C -1.2695,E1 24.9225,E2 208.715} C_DIS
LIN {X -68.7865,Y -116.5668,Z 156,A -124.5299,B 24.9708,C -1.2476,E1 24.9164,E2 211.2638} C_DIS
LIN {X -72.9268,Y -114.022,Z 156,A -125.9103,B 24.9691,C -1.2854,E1 24.9134,E2 212.5589} C_DIS
LIN {X -75.9503,Y -112.0308,Z 156,A -127.621,B 24.9694,C -1.2788,E1 24.9093,E2 214.2909} C_DIS
LIN {X -79.5713,Y -109.4887,Z 156,A -129.5061,B 24.9692,C -1.2814,E1 24.905,E2 216.1763} C_DIS
LIN {X -83.1725,Y -106.779,Z 156,A -131.4272,B 24.9692,C -1.2842,E1 24.9008,E2 218.0977} C_DIS
LIN {X -86.6777,Y -103.9542,Z 156,A -133.3712,B 24.969,C -1.2859,E1 24.8966,E2 220.0449} C_DIS
LIN {X -90.0647,Y -101.0335,Z 156,A -135.2592,B 24.9688,C -1.29,E1 24.8926,E2 221.9307} C_DIS
LIN {X -93.3611,Y -97.9953,Z 156,A -137.1055,B 24.9685,C -1.2966,E1 24.8889,E2 223.7689} C_DIS
LIN {X -96.5676,Y -94.8369,Z 156,A -139.0589,B 24.9685,C -1.2983,E1 24.885,E2 225.7264} C_DIS
LIN {X -99.5932,Y -91.6544,Z 156,A -140.9255,B 24.9682,C -1.3022,E1 24.8814,E2 227.592} C_DIS
LIN {X -102.6385,Y -88.2308,Z 156,A -142.845,B 24.968,C -1.3077,E1 24.8779,E2 229.507} C_DIS
LIN {X -105.3114,Y -85.0226,Z 156,A -144.6373,B 24.9678,C -1.3108,E1 24.8747,E2 231.3003} C_DIS
LIN {X -108.3882,Y -81.0642,Z 156,A -146.7944,B 24.9676,C -1.3143,E1 24.8711,E2 233.4593} C_DIS
LIN {X -110.9989,Y -77.4507,Z 156,A -148.6827,B 24.9674,C -1.3191,E1 24.868,E2 235.3454} C_DIS
LIN {X -113.389,Y -73.9075,Z 156,A -150.4995,B 24.9672,C -1.3235,E1 24.8652,E2 237.1609} C_DIS
LIN {X -115.665,Y -70.2925,Z 156,A -152.3407,B 24.967,C -1.3267,E1 24.8625,E2 239.0037} C_DIS
LIN {X -117.9298,Y -66.4222,Z 156,A -154.2363,B 24.9668,C -1.3321,E1 24.8599,E2 240.8964} C_DIS
LIN {X -119.9047,Y -62.7828,Z 156,A -155.9391,B 24.9664,C -1.3396,E1 24.8576,E2 242.5905} C_DIS
LIN {X -121.5173,Y -59.6023,Z 156,A -157.4024,B 24.9661,C -1.3462,E1 24.8558,E2 244.0459} C_DIS
LIN {X -122.9923,Y -56.496,Z 156,A -158.861,B 24.9658,C -1.3503,E1 24.8541,E2 245.5027} C_DIS
LIN {X -124.3197,Y -53.5115,Z 156,A -160.2634,B 24.9657,C -1.3534,E1 24.8525,E2 246.9054} C_DIS
LIN {X -125.605,Y -50.4206,Z 156,A -161.6874,B 24.9655,C -1.3573,E1 24.851,E2 248.3281} C_DIS
LIN {X -126.8375,Y -47.2348,Z 156,A -163.1524,B 24.9653,C -1.3607,E1 24.8496,E2 249.7932} C_DIS
LIN {X -127.876,Y -44.3458,Z 156,A -164.4863,B 24.9653,C -1.363,E1 24.8483,E2 251.1293} C_DIS
LIN {X -128.983,Y -41.0152,Z 156,A -165.9747,B 24.965,C -1.3674,E1 24.8471,E2 252.6156} C_DIS
LIN {X -130.0634,Y -37.453,Z 156,A -167.796,B 24.9653,C -1.3602,E1 24.8456,E2 254.4645} C_DIS
LIN {X -131.3025,Y -32.8442,Z 156,A -169.657,B 24.9646,C -1.3744,E1 24.8443,E2 256.3026} C_DIS
LIN {X -133.2601,Y -23.6785,Z 156,A -173.5566,B 24.9638,C -1.3904,E1 24.8421,E2 260.187} C_DIS
LIN {X -133.7976,Y -20.4249,Z 156,A -174.9652,B 24.9636,C -1.3943,E1 24.8415,E2 261.5949} C_DIS
LIN {X -134.3451,Y -16.4463,Z 156,A -176.7676,B 24.9636,C -1.3948,E1 24.8408,E2 263.4068} C_DIS
LIN {X -134.7517,Y -12.6875,Z 156,A -178.2849,B 24.9631,C -1.4041,E1 24.8404,E2 264.911} C_DIS
LIN {X -135.0636,Y -8.7721,Z 156,A 179.9449,B 24.9631,C -1.4043,E1 24.8401,E2 266.6914} C_DIS
LIN {X -135.2549,Y -5.0125,Z 156,A 178.3188,B 24.9629,C -1.408,E1 24.8399,E2 268.3185} C_DIS
LIN {X -135.345,Y -0.8709,Z 156,A 176.5843,B 24.9625,C -1.4147,E1 24.8398,E2 270.0474} C_DIS
LIN {X -135.3023,Y 3.5071,Z 156,A 174.7543,B 24.9621,C -1.422,E1 24.8398,E2 271.8711} C_DIS
LIN {X -135.1551,Y 7.2258,Z 156,A 173.1258,B 24.962,C -1.4246,E1 24.8401,E2 273.5031} C_DIS
LIN {X -134.8685,Y 11.3761,Z 156,A 171.4132,B 24.9615,C -1.4328,E1 24.8404,E2 275.2064} C_DIS
LIN {X -134.4911,Y 15.2191,Z 156,A 169.6815,B 24.9615,C -1.4335,E1 24.841,E2 276.947} C_DIS
LIN {X -133.9953,Y 19.0834,Z 156,A 168.1037,B 24.961,C -1.4425,E1 24.8415,E2 278.5128} C_DIS
LIN {X -133.433,Y 22.687,Z 156,A 166.4625,B 24.961,C -1.4428,E1 24.8423,E2 280.1629} C_DIS
LIN {X -132.6273,Y 26.9977,Z 156,A 164.697,B 24.9604,C -1.4533,E1 24.8432,E2 281.9138} C_DIS
LIN {X -131.5252,Y 31.9381,Z 156,A 162.5556,B 24.96,C -1.4604,E1 24.8446,E2 284.0508} C_DIS
LIN {X -130.7206,Y 35.086,Z 156,A 161.1068,B 24.96,C -1.4613,E1 24.8456,E2 285.506} C_DIS
LIN {X -129.5041,Y 39.3397,Z 156,A 158.6356,B 24.9613,C -1.4382,E1 24.8476,E2 288.0464} C_DIS
LIN {X -127.9587,Y 44.1074,Z 156,A 157.3603,B 24.9586,C -1.4863,E1 24.8487,E2 289.2144} C_DIS
LIN {X -126.6723,Y 47.6759,Z 156,A 155.4919,B 24.959,C -1.4785,E1 24.8505,E2 291.1121} C_DIS
LIN {X -125.4036,Y 50.9202,Z 156,A 154.0346,B 24.9587,C -1.484,E1 24.852,E2 292.5643} C_DIS
LIN {X -124.1173,Y 53.9795,Z 156,A 152.6222,B 24.9585,C -1.488,E1 24.8535,E2 293.975} C_DIS
LIN {X -122.7763,Y 56.9633,Z 156,A 151.2243,B 24.9583,C -1.4917,E1 24.8551,E2 295.3719} C_DIS
LIN {X -121.3056,Y 60.0314,Z 156,A 149.7887,B 24.9581,C -1.4963,E1 24.8569,E2 296.8042} C_DIS
LIN {X -119.2568,Y 64.009,Z 156,A 147.7994,B 24.958,C -1.4973,E1 24.8595,E2 298.8016} C_DIS
LIN {X -117.2114,Y 67.6819,Z 156,A 145.9656,B 24.9578,C -1.5,E1 24.862,E2 300.6387} C_DIS
LIN {X -114.8186,Y 71.6663,Z 156,A 143.9879,B 24.9576,C -1.5052,E1 24.8649,E2 302.614} C_DIS
LIN {X -112.3374,Y 75.4971,Z 156,A 142.0325,B 24.9573,C -1.5096,E1 24.8679,E2 304.5688} C_DIS
LIN {X -109.7958,Y 79.1475,Z 156,A 139.7489,B 24.9581,C -1.4953,E1 24.8717,E2 306.8977} C_DIS
LIN {X -107.1852,Y 82.6486,Z 156,A 138.4211,B 24.9564,C -1.526,E1 24.8738,E2 308.1588} C_DIS
LIN {X -104.8584,Y 85.5807,Z 156,A 136.7027,B 24.9565,C -1.5236,E1 24.8768,E2 309.8907} C_DIS
LIN {X -100.1486,Y 91.0473,Z 156,A 133.488,B 24.9565,C -1.5237,E1 24.8828,E2 313.1197} C_DIS
LIN {X -96.197,Y 95.213,Z 156,A 131.1962,B 24.9558,C -1.5367,E1 24.8872,E2 315.3904} C_DIS
LIN {X -93.0999,Y 98.2437,Z 156,A 129.2048,B 24.9559,C -1.5334,E1 24.8912,E2 317.3981} C_DIS
LIN {X -88.6316,Y 102.2934,Z 156,A 127.0465,B 24.9545,C -1.559,E1 24.8956,E2 319.504} C_DIS
LIN {X -86.5489,Y 104.061,Z 156,A 125.6072,B 24.9551,C -1.5475,E1 24.8988,E2 320.976} C_DIS
LIN {X -83.2083,Y 106.7513,Z 156,A 123.7672,B 24.955,C -1.5503,E1 24.9028,E2 322.8163} C_DIS
LIN {X -78.1711,Y 110.4928,Z 156,A 121.4705,B 24.9536,C -1.574,E1 24.9079,E2 325.0649} C_DIS
LIN {X -75.8035,Y 112.1301,Z 156,A 119.7114,B 24.955,C -1.5494,E1 24.9121,E2 326.8884} C_DIS
LIN {X -73.1134,Y 113.9025,Z 156,A 118.3199,B 24.955,C -1.5506,E1 24.9153,E2 328.2813} C_DIS
LIN {X -70.2781,Y 115.6736,Z 156,A 117.1021,B 24.9542,C -1.5632,E1 24.9182,E2 329.4731} C_DIS
LIN {X -66.4523,Y 117.9129,Z 156,A 115.2163,B 24.954,C -1.5661,E1 24.9227,E2 331.3574} C_DIS
LIN {X -62.6816,Y 119.9578,Z 156,A 113.4974,B 24.9536,C -1.5742,E1 24.9269,E2 333.0621} C_DIS
LIN {X -59.6109,Y 121.513,Z 156,A 112.0403,B 24.9534,C -1.5766,E1 24.9306,E2 334.5173} C_DIS
LIN {X -56.5037,Y 122.9888,Z 156,A 110.5888,B 24.9533,C -1.5791,E1 24.9342,E2 335.9664} C_DIS
LIN {X -53.4688,Y 124.3381,Z 156,A 109.184,B 24.9531,C -1.5813,E1 24.9378,E2 337.3694} C_DIS
LIN {X -50.3574,Y 125.6305,Z 156,A 107.7534,B 24.9531,C -1.5831,E1 24.9415,E2 338.7988} C_DIS
LIN {X -47.449,Y 126.7573,Z 156,A 106.4325,B 24.9529,C -1.5849,E1 24.9449,E2 340.1183} C_DIS
LIN {X -44.2387,Y 127.9132,Z 156,A 104.976,B 24.9529,C -1.5862,E1 24.9488,E2 341.5746} C_DIS
LIN {X -41.0402,Y 128.975,Z 156,A 103.5321,B 24.9529,C -1.587,E1 24.9526,E2 343.0192} C_DIS
LIN {X -37.7876,Y 129.9654,Z 156,A 102.086,B 24.9527,C -1.5883,E1 24.9565,E2 344.4646} C_DIS
LIN {X -33.7528,Y 131.0718,Z 156,A 100.2596,B 24.9527,C -1.5873,E1 24.9614,E2 346.2962} C_DIS
LIN {X -30.292,Y 131.9139,Z 156,A 98.7707,B 24.9527,C -1.5897,E1 24.9655,E2 347.7813} C_DIS
LIN {X -26.8319,Y 132.661,Z 156,A 97.3154,B 24.9524,C -1.5932,E1 24.9694,E2 349.23} C_DIS
LIN {X -23.5746,Y 133.2786,Z 156,A 95.9343,B 24.9524,C -1.5955,E1 24.9732,E2 350.6072} C_DIS
LIN {X -20.4959,Y 133.7866,Z 156,A 94.5762,B 24.9524,C -1.5945,E1 24.977,E2 351.9689} C_DIS
LIN {X -16.3847,Y 134.3524,Z 156,A 92.7813,B 24.9524,C -1.5936,E1 24.9819,E2 353.7672} C_DIS
LIN {X -12.8133,Y 134.7396,Z 156,A 91.3046,B 24.9522,C -1.5967,E1 24.986,E2 355.2374} C_DIS
LIN {X -9.2011,Y 135.0359,Z 156,A 89.6302,B 24.9526,C -1.5901,E1 24.9907,E2 356.9281} C_DIS
LIN {X -5.1133,Y 135.251,Z 156,A 88.01,B 24.9522,C -1.5966,E1 24.9952,E2 358.5333} C_DIS
LIN {X -0.9551,Y 135.3443,Z 156,A 86.2441,B 24.9522,C -1.5968,E1 25.0001,E2 360.299} C_DIS
LIN {X 2.4839,Y 135.3249,Z 156,A 84.7952,B 24.9522,C -1.5973,E1 25.0042,E2 361.7463} C_DIS
LIN {X 6.6072,Y 135.1862,Z 156,A 83.0212,B 24.9522,C -1.596,E1 25.0091,E2 363.5229} C_DIS
LIN {X 10.5952,Y 134.9341,Z 156,A 81.244,B 24.9525,C -1.5915,E1 25.0141,E2 365.3101} C_DIS
LIN {X 14.5035,Y 134.5681,Z 156,A 79.6821,B 24.9522,C -1.5965,E1 25.0184,E2 366.8592} C_DIS
LIN {X 18.6917,Y 134.0512,Z 156,A 77.85,B 24.9524,C -1.5937,E1 25.0235,E2 368.6964} C_DIS
LIN {X 22.3535,Y 133.4886,Z 156,A 76.3517,B 24.9522,C -1.5968,E1 25.0276,E2 370.1858} C_DIS
LIN {X 25.5679,Y 132.9105,Z 156,A 74.9554,B 24.9522,C -1.5955,E1 25.0315,E2 371.5836} C_DIS
LIN {X 29.3558,Y 132.1278,Z 156,A 73.1608,B 24.9528,C -1.5864,E1 25.0364,E2 373.3975} C_DIS
LIN {X 33.2695,Y 131.1945,Z 156,A 71.6239,B 24.9524,C -1.5942,E1 25.0405,E2 374.9137} C_DIS
LIN {X 36.5117,Y 130.3294,Z 156,A 70.1954,B 24.9524,C -1.5928,E1 25.0444,E2 376.3432} C_DIS
LIN {X 40.163,Y 129.2521,Z 156,A 68.6539,B 24.9524,C -1.5953,E1 25.0485,E2 377.8761} C_DIS
LIN {X 43.1496,Y 128.2853,Z 156,A 67.1762,B 24.9529,C -1.5862,E1 25.0524,E2 379.3724} C_DIS
LIN {X 47.7115,Y 126.659,Z 156,A 65.2416,B 24.9526,C -1.5904,E1 25.0575,E2 381.293} C_DIS
LIN {X 50.7868,Y 125.4574,Z 156,A 63.8262,B 24.9527,C -1.5881,E1 25.0612,E2 382.7108} C_DIS
LIN {X 53.967,Y 124.1227,Z 156,A 62.3906,B 24.9527,C -1.5877,E1 25.0648,E2 384.1438} C_DIS
LIN {X 57.0112,Y 122.7541,Z 156,A 60.9644,B 24.9529,C -1.5853,E1 25.0685,E2 385.5721} C_DIS
LIN {X 60.1015,Y 121.2711,Z 156,A 59.5249,B 24.9529,C -1.5841,E1 25.0721,E2 387.0107} C_DIS
LIN {X 63.1985,Y 119.6864,Z 156,A 58.0226,B 24.9532,C -1.5805,E1 25.0758,E2 388.5173} C_DIS
LIN {X 66.8226,Y 117.7037,Z 156,A 55.9533,B 24.9544,C -1.5607,E1 25.0809,E2 390.6272} C_DIS
LIN {X 69.935,Y 115.8812,Z 156,A 54.8558,B 24.9531,C -1.5815,E1 25.0835,E2 391.6722} C_DIS
LIN {X 73.1207,Y 113.8979,Z 156,A 53.1185,B 24.9538,C -1.5709,E1 25.0876,E2 393.4289} C_DIS
LIN {X 76.8667,Y 111.4044,Z 156,A 51.2037,B 24.954,C -1.5672,E1 25.092,E2 395.3462} C_DIS
LIN {X 80.5062,Y 108.8037,Z 156,A 49.3202,B 24.9542,C -1.5643,E1 25.0963,E2 397.2298} C_DIS
LIN {X 84.3316,Y 105.8655,Z 156,A 47.089,B 24.955,C -1.5502,E1 25.1012,E2 399.486} C_DIS
LIN {X 86.8971,Y 103.7701,Z 156,A 46.0714,B 24.9539,C -1.5684,E1 25.1033,E2 400.4568} C_DIS
LIN {X 89.7026,Y 101.3547,Z 156,A 44.3545,B 24.9546,C -1.557,E1 25.107,E2 402.1937} C_DIS
LIN {X 93.0196,Y 98.3195,Z 156,A 42.4446,B 24.9548,C -1.5527,E1 25.1109,E2 404.1061} C_DIS
LIN {X 96.0747,Y 95.3361,Z 156,A 40.648,B 24.955,C -1.5493,E1 25.1145,E2 405.903} C_DIS
LIN {X 99.2364,Y 92.041,Z 156,A 38.7609,B 24.9551,C -1.5474,E1 25.1181,E2 407.7863} C_DIS
LIN {X 102.0805,Y 88.8759,Z 156,A 36.9351,B 24.9555,C -1.5419,E1 25.1215,E2 409.6171} C_DIS
LIN {X 104.892,Y 85.5395,Z 156,A 35.0837,B 24.9557,C -1.5372,E1 25.1248,E2 411.4711} C_DIS
LIN {X 107.7305,Y 81.9365,Z 156,A 33.1407,B 24.956,C -1.5322,E1 25.1281,E2 413.4166} C_DIS
LIN {X 110.935,Y 77.5421,Z 156,A 30.5384,B 24.9573,C -1.5098,E1 25.1324,E2 416.0591} C_DIS
LIN {X 113.1633,Y 74.2525,Z 156,A 29.2138,B 24.9564,C -1.525,E1 25.1344,E2 417.3412} C_DIS
LIN {X 115.5704,Y 70.4482,Z 156,A 27.2891,B 24.9568,C -1.5188,E1 25.1372,E2 419.2708} C_DIS
LIN {X 117.9107,Y 66.4562,Z 156,A 25.3362,B 24.9571,C -1.5137,E1 25.1399,E2 421.2256} C_DIS
LIN {X 120.0025,Y 62.5965,Z 156,A 23.6369,B 24.9569,C -1.5174,E1 25.1421,E2 422.9074} C_DIS
LIN {X 122.6302,Y 57.2793,Z 156,A 21.2278,B 24.9569,C -1.5157,E1 25.1451,E2 425.3074} C_DIS
LIN {X 124.3198,Y 53.511,Z 156,A 19.3767,B 24.9576,C -1.5049,E1 25.1472,E2 427.1741} C_DIS
LIN {X 125.7115,Y 50.1564,Z 156,A 17.841,B 24.9578,C -1.5003,E1 25.1488,E2 428.712} C_DIS
LIN {X 127.1673,Y 46.3414,Z 156,A 15.9766,B 24.9585,C -1.4875,E1 25.1506,E2 430.5962} C_DIS
LIN {X 128.4995,Y 42.5064,Z 156,A 14.3684,B 24.9585,C -1.4884,E1 25.1521,E2 432.1932} C_DIS
LIN {X 130.0514,Y 37.494,Z 156,A 12.2395,B 24.9585,C -1.4866,E1 25.1538,E2 434.3142} C_DIS
LIN {X 130.8522,Y 34.5926,Z 156,A 10.9711,B 24.9588,C -1.483,E1 25.1547,E2 435.5839} C_DIS
LIN {X 131.6302,Y 31.5023,Z 156,A 9.5607,B 24.9592,C -1.4752,E1 25.1557,E2 437.0044} C_DIS
LIN {X 132.6123,Y 27.0715,Z 156,A 7.699,B 24.9594,C -1.4724,E1 25.1568,E2 438.8619} C_DIS
LIN {X 133.237,Y 23.8073,Z 156,A 6.2885,B 24.9596,C -1.4677,E1 25.1575,E2 440.2752} C_DIS
LIN {X 133.7894,Y 20.478,Z 156,A 4.8945,B 24.9598,C -1.465,E1 25.1581,E2 441.6674} C_DIS
LIN {X 134.2416,Y 17.2683,Z 156,A 3.422,B 24.9603,C -1.4549,E1 25.1586,E2 443.1551} C_DIS
LIN {X 134.7021,Y 13.2033,Z 156,A 1.7397,B 24.9605,C -1.452,E1 25.1591,E2 444.8342} C_DIS
LIN {X 135.0127,Y 9.5197,Z 156,A 0.1224,B 24.9609,C -1.4439,E1 25.1595,E2 446.461} C_DIS
LIN {X 135.2462,Y 5.2344,Z 156,A -1.559,B 24.9609,C -1.4455,E1 25.1597,E2 448.1286} C_DIS
LIN {X 135.343,Y 1.2521,Z 156,A -3.3389,B 24.9614,C -1.4346,E1 25.1597,E2 449.9235} C_DIS
LIN {X 135.3158,Y -3.0198,Z 156,A -5.163,B 24.9618,C -1.4277,E1 25.1597,E2 451.7531} C_DIS
LIN {X 135.1672,Y -6.9869,Z 156,A -6.744,B 24.9618,C -1.4277,E1 25.1595,E2 453.3245} C_DIS
LIN {X 134.8673,Y -11.3905,Z 156,A -8.5391,B 24.9619,C -1.4257,E1 25.1591,E2 455.1139} C_DIS
LIN {X 134.5328,Y -14.8309,Z 156,A -10.0159,B 24.9622,C -1.4201,E1 25.1587,E2 456.5952} C_DIS
LIN {X 134.0195,Y -18.9136,Z 156,A -11.7881,B 24.9626,C -1.4126,E1 25.1581,E2 458.3746} C_DIS
LIN {X 133.4455,Y -22.6121,Z 156,A -13.2792,B 24.9626,C -1.4126,E1 25.1574,E2 459.8569} C_DIS
LIN {X 132.8198,Y -26.0423,Z 156,A -14.8576,B 24.9632,C -1.4019,E1 25.1566,E2 461.4512} C_DIS
LIN {X 131.9849,Y -29.9812,Z 156,A -16.5076,B 24.9633,C -1.3994,E1 25.1556,E2 463.0975} C_DIS
LIN {X 131.1682,Y -33.3733,Z 156,A -17.9402,B 24.9634,C -1.3971,E1 25.1546,E2 464.5273} C_DIS
LIN {X 130.2948,Y -36.6353,Z 156,A -19.3621,B 24.9637,C -1.3929,E1 25.1536,E2 465.951} C_DIS
LIN {X 129.1975,Y -40.3413,Z 156,A -21.1291,B 24.9643,C -1.3802,E1 25.1521,E2 467.7378} C_DIS
LIN {X 128.0209,Y -43.928,Z 156,A -22.6279,B 24.9643,C -1.3806,E1 25.1508,E2 469.2271} C_DIS
LIN {X 126.3343,Y -48.5666,Z 156,A -24.5217,B 24.9641,C -1.385,E1 25.149,E2 471.1} C_DIS
LIN {X 124.7782,Y -52.4338,Z 156,A -26.533,B 24.9651,C -1.3655,E1 25.1468,E2 473.1462} C_DIS
LIN {X 122.726,Y -57.0719,Z 156,A -28.5227,B 24.965,C -1.3677,E1 25.1446,E2 475.1199} C_DIS
LIN {X 121.2452,Y -60.1539,Z 156,A -30.002,B 24.9653,C -1.3614,E1 25.1427,E2 476.6061} C_DIS
LIN {X 119.2787,Y -63.9682,Z 156,A -31.8085,B 24.9655,C -1.3564,E1 25.1404,E2 478.4148} C_DIS
LIN {X 117.3079,Y -67.5153,Z 156,A -33.5848,B 24.966,C -1.348,E1 25.1379,E2 480.2018} C_DIS
LIN {X 115.1198,Y -71.1823,Z 156,A -35.3195,B 24.966,C -1.3468,E1 25.1354,E2 481.9305} C_DIS
LIN {X 113.0375,Y -74.4437,Z 156,A -36.9728,B 24.9663,C -1.3411,E1 25.1329,E2 483.5888} C_DIS
LIN {X 110.6552,Y -77.9407,Z 156,A -38.7817,B 24.9666,C -1.335,E1 25.13,E2 485.4032} C_DIS
LIN {X 106.6974,Y -83.2775,Z 156,A -41.5979,B 24.967,C -1.327,E1 25.1253,E2 488.225} C_DIS
LIN {X 103.9153,Y -86.724,Z 156,A -43.4763,B 24.9673,C -1.3217,E1 25.122,E2 490.1071} C_DIS
LIN {X 101.0529,Y -90.0431,Z 156,A -45.3301,B 24.9675,C -1.3169,E1 25.1185,E2 491.964} C_DIS
LIN {X 97.6302,Y -93.7424,Z 156,A -47.3751,B 24.9675,C -1.3163,E1 25.1146,E2 494.0013} C_DIS
LIN {X 95.1635,Y -96.2462,Z 156,A -48.9052,B 24.9678,C -1.3102,E1 25.1116,E2 495.5393} C_DIS
LIN {X 91.9016,Y -99.3659,Z 156,A -50.7878,B 24.968,C -1.3071,E1 25.1078,E2 497.4216} C_DIS
Enddeposition()
END
